LIN {X 0,Y 573.653,Z 410.287,A -85,B 0,C 180,E1 -2261.447,E2 -2261.447} C_VEL
LIN {X 0,Y 573.725,Z 397.169,A -85,B 0,C 180,E1 -2261.975,E2 -2261.975} C_VEL
LIN {X 0,Y 573.84,Z 384.516,A -85,B 0,C 180,E1 -2262.331,E2 -2262.331} C_VEL
LIN {X 0,Y 573.891,Z 371.307,A -85,B 0,C 180,E1 -2262.555,E2 -2262.555} C_VEL
LIN {X 0,Y 573.878,Z 274.271,A -85,B 0,C 180,E1 -2263.777,E2 -2263.777} C_VEL
LIN {X 0,Y 573.4,Z 270.792,A -85,B 0,C 180,E1 -2263.85,E2 -2263.85} C_VEL
LIN {X 0,Y 573.536,Z 250.898,A -85,B 0,C 180,E1 -2266.722,E2 -2266.722} C_VEL
LIN {X 0,Y 573.751,Z 233.17,A -85,B 0,C 180,E1 -2269.313,E2 -2269.313} C_VEL
LIN {X 0,Y 573.937,Z 214.032,A -85,B 0,C 180,E1 -2272.12,E2 -2272.12} C_VEL
LIN {X 0,Y 573.619,Z 210.185,A -85,B 0,C 180,E1 -2272.702,E2 -2272.702} C_VEL
LIN {X 0,Y 573.234,Z 208.084,A -85,B 0,C 180,E1 -2273.06,E2 -2273.06} C_VEL
LIN {X 0,Y 573.236,Z 208.085,A -85,B 0,C 180,E1 -2275.411,E2 -2275.411} C_VEL
LIN {X 0,Y 573.231,Z 208.076,A -85,B 0,C 180,E1 -2278.565,E2 -2278.565} C_VEL
LIN {X 0,Y 573.22,Z 208.08,A -85,B 0,C 180,E1 -2280.994,E2 -2280.994} C_VEL
LIN {X 0,Y 573.265,Z 208.081,A -85,B 0,C 180,E1 -2283.524,E2 -2283.524} C_VEL
LIN {X 0,Y 573.194,Z 208.082,A -85,B 0,C 180,E1 -2286.053,E2 -2286.053} C_VEL
LIN {X 0,Y 573.237,Z 208.075,A -85,B 0,C 180,E1 -2288.702,E2 -2288.702} C_VEL
LIN {X 0,Y 573.226,Z 208.084,A -85,B 0,C 180,E1 -2291.592,E2 -2291.592} C_VEL
LIN {X 0,Y 573.223,Z 208.076,A -85,B 0,C 180,E1 -2294.335,E2 -2294.335} C_VEL
LIN {X 0,Y 573.237,Z 208.083,A -85,B 0,C 180,E1 -2297.359,E2 -2297.359} C_VEL
LIN {X 0,Y 573.237,Z 208.074,A -85,B 0,C 180,E1 -2300.392,E2 -2300.392} C_VEL
LIN {X 0,Y 573.226,Z 208.079,A -85,B 0,C 180,E1 -2303.075,E2 -2303.075} C_VEL
LIN {X 0,Y 573.262,Z 208.077,A -85,B 0,C 180,E1 -2305.671,E2 -2305.671} C_VEL
LIN {X 0,Y 573.239,Z 208.075,A -85,B 0,C 180,E1 -2308.184,E2 -2308.184} C_VEL
LIN {X 0,Y 573.26,Z 208.071,A -85,B 0,C 180,E1 -2310.634,E2 -2310.634} C_VEL
LIN {X 0,Y 573.255,Z 208.075,A -85,B 0,C 180,E1 -2313.81,E2 -2313.81} C_VEL
LIN {X 0,Y 573.227,Z 208.076,A -85,B 0,C 180,E1 -2316.134,E2 -2316.134} C_VEL
LIN {X 0,Y 573.251,Z 208.077,A -85,B 0,C 180,E1 -2319.174,E2 -2319.174} C_VEL
LIN {X 0,Y 573.221,Z 208.086,A -85,B 0,C 180,E1 -2321.411,E2 -2321.411} C_VEL
LIN {X 0,Y 573.242,Z 208.08,A -85,B 0,C 180,E1 -2323.621,E2 -2323.621} C_VEL
LIN {X 0,Y 573.273,Z 208.074,A -85,B 0,C 180,E1 -2325.807,E2 -2325.807} C_VEL
LIN {X 0,Y 573.265,Z 208.071,A -85,B 0,C 180,E1 -2328.745,E2 -2328.745} C_VEL
LIN {X 0,Y 573.283,Z 208.076,A -85,B 0,C 180,E1 -2331.541,E2 -2331.541} C_VEL
LIN {X 0,Y 573.246,Z 208.079,A -85,B 0,C 180,E1 -2333.665,E2 -2333.665} C_VEL
LIN {X 0,Y 573.229,Z 208.079,A -85,B 0,C 180,E1 -2335.781,E2 -2335.781} C_VEL
LIN {X 0,Y 573.314,Z 208.067,A -85,B 0,C 180,E1 -2337.892,E2 -2337.892} C_VEL
LIN {X 0,Y 573.319,Z 208.065,A -85,B 0,C 180,E1 -2340.702,E2 -2340.702} C_VEL
LIN {X 0,Y 573.292,Z 208.068,A -85,B 0,C 180,E1 -2342.811,E2 -2342.811} C_VEL
LIN {X 0,Y 573.293,Z 208.074,A -85,B 0,C 180,E1 -2345.628,E2 -2345.628} C_VEL
LIN {X 0,Y 573.253,Z 208.071,A -85,B 0,C 180,E1 -2348.46,E2 -2348.46} C_VEL
LIN {X 0,Y 573.274,Z 208.078,A -85,B 0,C 180,E1 -2351.312,E2 -2351.312} C_VEL
LIN {X 0,Y 573.27,Z 208.07,A -85,B 0,C 180,E1 -2354.419,E2 -2354.419} C_VEL
LIN {X 0,Y 573.251,Z 208.077,A -85,B 0,C 180,E1 -2357.112,E2 -2357.112} C_VEL
LIN {X 0,Y 573.238,Z 208.075,A -85,B 0,C 180,E1 -2360.077,E2 -2360.077} C_VEL
LIN {X 0,Y 573.225,Z 208.074,A -85,B 0,C 180,E1 -2362.338,E2 -2362.338} C_VEL
LIN {X 0,Y 573.221,Z 208.076,A -85,B 0,C 180,E1 -2364.362,E2 -2364.362} C_VEL
LIN {X 0,Y 572.579,Z 208.16,A -85,B 0,C 180,E1 -2364.948,E2 -2364.948} C_VEL
LIN {X 0,Y 569.74,Z 208.519,A -85,B 0,C 180,E1 -2365.899,E2 -2365.899} C_VEL
LIN {X 0,Y 567.321,Z 208.823,A -85,B 0,C 180,E1 -2366.665,E2 -2366.665} C_VEL
LIN {X 0,Y 566.272,Z 208.95,A -85,B 0,C 180,E1 -2367.256,E2 -2367.256} C_VEL
LIN {X 0,Y 566.183,Z 208.959,A -85,B 0,C 180,E1 -2367.456,E2 -2367.456} C_VEL
LIN {X 0,Y 566.197,Z 208.955,A -85,B 0,C 180,E1 -2369.769,E2 -2369.769} C_VEL
LIN {X 0,Y 566.202,Z 208.951,A -85,B 0,C 180,E1 -2372.43,E2 -2372.43} C_VEL
LIN {X 0,Y 566.179,Z 208.957,A -85,B 0,C 180,E1 -2374.989,E2 -2374.989} C_VEL
LIN {X 0,Y 566.193,Z 208.961,A -85,B 0,C 180,E1 -2377.461,E2 -2377.461} C_VEL
LIN {X 0,Y 566.208,Z 208.95,A -85,B 0,C 180,E1 -2380.199,E2 -2380.199} C_VEL
LIN {X 0,Y 566.198,Z 208.956,A -85,B 0,C 180,E1 -2383.055,E2 -2383.055} C_VEL
LIN {X 0,Y 566.161,Z 208.956,A -85,B 0,C 180,E1 -2386.053,E2 -2386.053} C_VEL
LIN {X 0,Y 566.173,Z 208.958,A -85,B 0,C 180,E1 -2388.86,E2 -2388.86} C_VEL
LIN {X 0,Y 566.211,Z 208.96,A -85,B 0,C 180,E1 -2391.442,E2 -2391.442} C_VEL
LIN {X 0,Y 566.152,Z 208.958,A -85,B 0,C 180,E1 -2394.307,E2 -2394.307} C_VEL
LIN {X 0,Y 566.208,Z 208.953,A -85,B 0,C 180,E1 -2396.897,E2 -2396.897} C_VEL
LIN {X 0,Y 566.182,Z 208.962,A -85,B 0,C 180,E1 -2399.407,E2 -2399.407} C_VEL
LIN {X 0,Y 566.19,Z 208.956,A -85,B 0,C 180,E1 -2401.856,E2 -2401.856} C_VEL
LIN {X 0,Y 566.221,Z 209.027,A -85,B 0,C 180,E1 -2404.227,E2 -2404.227} C_VEL
LIN {X 0,Y 566.522,Z 213.688,A -85,B 0,C 180,E1 -2405.052,E2 -2405.052} C_VEL
LIN {X 0,Y 566.362,Z 230.218,A -85,B 0,C 180,E1 -2407.953,E2 -2407.953} C_VEL
LIN {X 0,Y 566.25,Z 242.171,A -85,B 0,C 180,E1 -2410.048,E2 -2410.048} C_VEL
LIN {X 0,Y 567.167,Z 248.554,A -85,B 0,C 180,E1 -2410.157,E2 -2410.157} C_VEL
LIN {X 0,Y 566.907,Z 349.31,A -85,B 0,C 180,E1 -2411.454,E2 -2411.454} C_VEL
LIN {X 0,Y 566.825,Z 362.732,A -85,B 0,C 180,E1 -2411.779,E2 -2411.779} C_VEL
LIN {X 0,Y 566.717,Z 375.02,A -85,B 0,C 180,E1 -2412.219,E2 -2412.219} C_VEL
LIN {X 0,Y 566.602,Z 386.826,A -85,B 0,C 180,E1 -2412.791,E2 -2412.791} C_VEL
LIN {X 0,Y 566.464,Z 398.37,A -85,B 0,C 180,E1 -2413.513,E2 -2413.513} C_VEL
LIN {X 0,Y 566.3,Z 408.957,A -85,B 0,C 180,E1 -2414.34,E2 -2414.34} C_VEL
LIN {X 0,Y 566.194,Z 418.423,A -85,B 0,C 180,E1 -2415.259,E2 -2415.259} C_VEL
LIN {X 0,Y 566.087,Z 427.544,A -85,B 0,C 180,E1 -2416.356,E2 -2416.356} C_VEL
LIN {X 0,Y 566.031,Z 434.851,A -85,B 0,C 180,E1 -2417.45,E2 -2417.45} C_VEL
LIN {X 0,Y 565.952,Z 440.637,A -85,B 0,C 180,E1 -2418.54,E2 -2418.54} C_VEL
LIN {X 0,Y 565.906,Z 445.169,A -85,B 0,C 180,E1 -2419.626,E2 -2419.626} C_VEL
LIN {X 0,Y 565.863,Z 448.594,A -85,B 0,C 180,E1 -2420.708,E2 -2420.708} C_VEL
LIN {X 0,Y 565.86,Z 450.288,A -85,B 0,C 180,E1 -2421.429,E2 -2421.429} C_VEL
LIN {X 0,Y 565.879,Z 451.573,A -85,B 0,C 180,E1 -2422.148,E2 -2422.148} C_VEL
LIN {X 0,Y 565.919,Z 452.869,A -85,B 0,C 180,E1 -2423.466,E2 -2423.466} C_VEL
LIN {X 0,Y 565.897,Z 452.951,A -85,B 0,C 180,E1 -2424.298,E2 -2424.298} C_VEL
LIN {X 0,Y 565.911,Z 451.892,A -85,B 0,C 180,E1 -2425.727,E2 -2425.727} C_VEL
LIN {X 0,Y 565.912,Z 450.734,A -85,B 0,C 180,E1 -2426.44,E2 -2426.44} C_VEL
LIN {X 0,Y 565.876,Z 449.165,A -85,B 0,C 180,E1 -2427.152,E2 -2427.152} C_VEL
LIN {X 0,Y 565.906,Z 446.016,A -85,B 0,C 180,E1 -2428.221,E2 -2428.221} C_VEL
LIN {X 0,Y 565.9,Z 441.822,A -85,B 0,C 180,E1 -2429.288,E2 -2429.288} C_VEL
LIN {X 0,Y 566.026,Z 435.459,A -85,B 0,C 180,E1 -2430.534,E2 -2430.534} C_VEL
LIN {X 0,Y 566.067,Z 428.544,A -85,B 0,C 180,E1 -2431.601,E2 -2431.601} C_VEL
LIN {X 0,Y 566.142,Z 419.905,A -85,B 0,C 180,E1 -2432.668,E2 -2432.668} C_VEL
LIN {X 0,Y 566.241,Z 411.087,A -85,B 0,C 180,E1 -2433.558,E2 -2433.558} C_VEL
LIN {X 0,Y 566.404,Z 400.228,A -85,B 0,C 180,E1 -2434.448,E2 -2434.448} C_VEL
LIN {X 0,Y 566.585,Z 389.269,A -85,B 0,C 180,E1 -2435.16,E2 -2435.16} C_VEL
LIN {X 0,Y 566.686,Z 377.045,A -85,B 0,C 180,E1 -2435.783,E2 -2435.783} C_VEL
LIN {X 0,Y 566.844,Z 365.434,A -85,B 0,C 180,E1 -2436.228,E2 -2436.228} C_VEL
LIN {X 0,Y 566.944,Z 352.308,A -85,B 0,C 180,E1 -2436.575,E2 -2436.575} C_VEL
LIN {X 0,Y 567.009,Z 333.787,A -85,B 0,C 180,E1 -2436.85,E2 -2436.85} C_VEL
LIN {X 0,Y 567.123,Z 247.443,A -85,B 0,C 180,E1 -2437.948,E2 -2437.948} C_VEL
LIN {X 0,Y 566.253,Z 242.163,A -85,B 0,C 180,E1 -2438.043,E2 -2438.043} C_VEL
LIN {X 0,Y 566.444,Z 224.855,A -85,B 0,C 180,E1 -2441.083,E2 -2441.083} C_VEL
LIN {X 0,Y 566.545,Z 211.416,A -85,B 0,C 180,E1 -2443.45,E2 -2443.45} C_VEL
LIN {X 0,Y 566.232,Z 208.954,A -85,B 0,C 180,E1 -2443.915,E2 -2443.915} C_VEL
LIN {X 0,Y 566.229,Z 208.952,A -85,B 0,C 180,E1 -2447.113,E2 -2447.113} C_VEL
LIN {X 0,Y 566.206,Z 208.95,A -85,B 0,C 180,E1 -2449.581,E2 -2449.581} C_VEL
LIN {X 0,Y 566.196,Z 208.951,A -85,B 0,C 180,E1 -2451.862,E2 -2451.862} C_VEL
LIN {X 0,Y 566.222,Z 208.952,A -85,B 0,C 180,E1 -2455.03,E2 -2455.03} C_VEL
LIN {X 0,Y 566.176,Z 208.955,A -85,B 0,C 180,E1 -2457.341,E2 -2457.341} C_VEL
LIN {X 0,Y 566.203,Z 208.95,A -85,B 0,C 180,E1 -2459.769,E2 -2459.769} C_VEL
LIN {X 0,Y 566.205,Z 208.956,A -85,B 0,C 180,E1 -2462.429,E2 -2462.429} C_VEL
LIN {X 0,Y 566.182,Z 208.958,A -85,B 0,C 180,E1 -2464.989,E2 -2464.989} C_VEL
LIN {X 0,Y 566.194,Z 208.952,A -85,B 0,C 180,E1 -2467.461,E2 -2467.461} C_VEL
LIN {X 0,Y 566.209,Z 208.953,A -85,B 0,C 180,E1 -2470.199,E2 -2470.199} C_VEL
LIN {X 0,Y 566.199,Z 208.955,A -85,B 0,C 180,E1 -2473.054,E2 -2473.054} C_VEL
LIN {X 0,Y 566.195,Z 208.953,A -85,B 0,C 180,E1 -2476.049,E2 -2476.049} C_VEL
LIN {X 0,Y 566.205,Z 208.952,A -85,B 0,C 180,E1 -2479.214,E2 -2479.214} C_VEL
LIN {X 0,Y 566.183,Z 208.953,A -85,B 0,C 180,E1 -2481.636,E2 -2481.636} C_VEL
LIN {X 0,Y 566.151,Z 208.961,A -85,B 0,C 180,E1 -2484.307,E2 -2484.307} C_VEL
LIN {X 0,Y 566.221,Z 208.954,A -85,B 0,C 180,E1 -2486.898,E2 -2486.898} C_VEL
LIN {X 0,Y 566.18,Z 208.954,A -85,B 0,C 180,E1 -2489.407,E2 -2489.407} C_VEL
LIN {X 0,Y 566.192,Z 208.952,A -85,B 0,C 180,E1 -2491.856,E2 -2491.856} C_VEL
LIN {X 0,Y 566.196,Z 208.955,A -85,B 0,C 180,E1 -2494.25,E2 -2494.25} C_VEL
LIN {X 0,Y 566.171,Z 208.963,A -85,B 0,C 180,E1 -2496.719,E2 -2496.719} C_VEL
LIN {X 0,Y 566.205,Z 208.95,A -85,B 0,C 180,E1 -2499.662,E2 -2499.662} C_VEL
LIN {X 0,Y 566.2,Z 208.961,A -85,B 0,C 180,E1 -2502.668,E2 -2502.668} C_VEL
LIN {X 0,Y 566.222,Z 208.948,A -85,B 0,C 180,E1 -2505.626,E2 -2505.626} C_VEL
LIN {X 0,Y 566.236,Z 208.956,A -85,B 0,C 180,E1 -2508.675,E2 -2508.675} C_VEL
LIN {X 0,Y 566.204,Z 208.95,A -85,B 0,C 180,E1 -2511.434,E2 -2511.434} C_VEL
LIN {X 0,Y 566.262,Z 208.948,A -85,B 0,C 180,E1 -2514.302,E2 -2514.302} C_VEL
LIN {X 0,Y 566.282,Z 208.941,A -85,B 0,C 180,E1 -2517.866,E2 -2517.866} C_VEL
LIN {X 0,Y 566.302,Z 208.947,A -85,B 0,C 180,E1 -2520.711,E2 -2520.711} C_VEL
LIN {X 0,Y 566.27,Z 208.948,A -85,B 0,C 180,E1 -2522.846,E2 -2522.846} C_VEL
LIN {X 0,Y 566.25,Z 208.945,A -85,B 0,C 180,E1 -2525.698,E2 -2525.698} C_VEL
LIN {X 0,Y 566.226,Z 208.957,A -85,B 0,C 180,E1 -2528.566,E2 -2528.566} C_VEL
LIN {X 0,Y 566.243,Z 208.945,A -85,B 0,C 180,E1 -2531.454,E2 -2531.454} C_VEL
LIN {X 0,Y 566.235,Z 208.955,A -85,B 0,C 180,E1 -2534.506,E2 -2534.506} C_VEL
LIN {X 0,Y 566.194,Z 208.952,A -85,B 0,C 180,E1 -2537.332,E2 -2537.332} C_VEL
LIN {X 0,Y 566.207,Z 208.956,A -85,B 0,C 180,E1 -2540.337,E2 -2540.337} C_VEL
LIN {X 0,Y 566.169,Z 208.955,A -85,B 0,C 180,E1 -2543.281,E2 -2543.281} C_VEL
LIN {X 0,Y 566.205,Z 208.95,A -85,B 0,C 180,E1 -2545.749,E2 -2545.749} C_VEL
LIN {X 0,Y 566.185,Z 208.957,A -85,B 0,C 180,E1 -2548.954,E2 -2548.954} C_VEL
LIN {X 0,Y 566.192,Z 208.952,A -85,B 0,C 180,E1 -2551.422,E2 -2551.422} C_VEL
LIN {X 0,Y 566.201,Z 208.952,A -85,B 0,C 180,E1 -2553.957,E2 -2553.957} C_VEL
LIN {X 0,Y 566.182,Z 208.963,A -85,B 0,C 180,E1 -2556.571,E2 -2556.571} C_VEL
LIN {X 0,Y 566.212,Z 208.95,A -85,B 0,C 180,E1 -2559.274,E2 -2559.274} C_VEL
LIN {X 0,Y 566.188,Z 208.955,A -85,B 0,C 180,E1 -2562.09,E2 -2562.09} C_VEL
LIN {X 0,Y 566.165,Z 208.958,A -85,B 0,C 180,E1 -2565.037,E2 -2565.037} C_VEL
LIN {X 0,Y 566.187,Z 208.954,A -85,B 0,C 180,E1 -2567.91,E2 -2567.91} C_VEL
LIN {X 0,Y 566.211,Z 208.956,A -85,B 0,C 180,E1 -2570.726,E2 -2570.726} C_VEL
LIN {X 0,Y 566.182,Z 208.953,A -85,B 0,C 180,E1 -2573.429,E2 -2573.429} C_VEL
LIN {X 0,Y 566.213,Z 208.955,A -85,B 0,C 180,E1 -2576.266,E2 -2576.266} C_VEL
LIN {X 0,Y 566.186,Z 208.956,A -85,B 0,C 180,E1 -2578.925,E2 -2578.925} C_VEL
LIN {X 0,Y 566.192,Z 208.954,A -85,B 0,C 180,E1 -2581.856,E2 -2581.856} C_VEL
LIN {X 0,Y 566.196,Z 208.958,A -85,B 0,C 180,E1 -2584.25,E2 -2584.25} C_VEL
LIN {X 0,Y 566.21,Z 209.141,A -85,B 0,C 180,E1 -2586.852,E2 -2586.852} C_VEL
LIN {X 0,Y 567.008,Z 213.862,A -85,B 0,C 180,E1 -2587.596,E2 -2587.596} C_VEL
LIN {X 0,Y 566.766,Z 233.934,A -85,B 0,C 180,E1 -2590.578,E2 -2590.578} C_VEL
LIN {X 0,Y 566.551,Z 252.227,A -85,B 0,C 180,E1 -2593.262,E2 -2593.262} C_VEL
LIN {X 0,Y 566.418,Z 271.144,A -85,B 0,C 180,E1 -2595.998,E2 -2595.998} C_VEL
LIN {X 0,Y 567.165,Z 276.51,A -85,B 0,C 180,E1 -2596.086,E2 -2596.086} C_VEL
LIN {X 0,Y 566.918,Z 378.947,A -85,B 0,C 180,E1 -2597.402,E2 -2597.402} C_VEL
LIN {X 0,Y 566.839,Z 392.218,A -85,B 0,C 180,E1 -2597.719,E2 -2597.719} C_VEL
LIN {X 0,Y 566.724,Z 404.378,A -85,B 0,C 180,E1 -2598.148,E2 -2598.148} C_VEL
LIN {X 0,Y 566.603,Z 416.367,A -85,B 0,C 180,E1 -2598.72,E2 -2598.72} C_VEL
LIN {X 0,Y 566.45,Z 428.197,A -85,B 0,C 180,E1 -2599.455,E2 -2599.455} C_VEL
LIN {X 0,Y 566.324,Z 438.604,A -85,B 0,C 180,E1 -2600.265,E2 -2600.265} C_VEL
LIN {X 0,Y 566.207,Z 447.113,A -85,B 0,C 180,E1 -2601.074,E2 -2601.074} C_VEL
LIN {X 0,Y 566.112,Z 454.961,A -85,B 0,C 180,E1 -2601.972,E2 -2601.972} C_VEL
LIN {X 0,Y 566.003,Z 462.622,A -85,B 0,C 180,E1 -2603.047,E2 -2603.047} C_VEL
LIN {X 0,Y 566.004,Z 469.68,A -85,B 0,C 180,E1 -2604.299,E2 -2604.299} C_VEL
LIN {X 0,Y 565.933,Z 474.373,A -85,B 0,C 180,E1 -2605.37,E2 -2605.37} C_VEL
LIN {X 0,Y 565.927,Z 477.958,A -85,B 0,C 180,E1 -2606.44,E2 -2606.44} C_VEL
LIN {X 0,Y 565.878,Z 479.808,A -85,B 0,C 180,E1 -2607.152,E2 -2607.152} C_VEL
LIN {X 0,Y 565.846,Z 482.184,A -85,B 0,C 180,E1 -2608.577,E2 -2608.577} C_VEL
LIN {X 0,Y 565.839,Z 483,A -85,B 0,C 180,E1 -2610,E2 -2610} C_VEL
LIN {X 0,Y 565.846,Z 482.185,A -85,B 0,C 180,E1 -2611.423,E2 -2611.423} C_VEL
LIN {X 0,Y 565.878,Z 479.81,A -85,B 0,C 180,E1 -2612.848,E2 -2612.848} C_VEL
LIN {X 0,Y 565.926,Z 476.895,A -85,B 0,C 180,E1 -2613.917,E2 -2613.917} C_VEL
LIN {X 0,Y 565.878,Z 472.948,A -85,B 0,C 180,E1 -2614.987,E2 -2614.987} C_VEL
LIN {X 0,Y 566.002,Z 467.867,A -85,B 0,C 180,E1 -2616.059,E2 -2616.059} C_VEL
LIN {X 0,Y 566.04,Z 461.467,A -85,B 0,C 180,E1 -2617.132,E2 -2617.132} C_VEL
LIN {X 0,Y 566.134,Z 453.477,A -85,B 0,C 180,E1 -2618.208,E2 -2618.208} C_VEL
LIN {X 0,Y 566.229,Z 445.334,A -85,B 0,C 180,E1 -2619.105,E2 -2619.105} C_VEL
LIN {X 0,Y 566.345,Z 435.399,A -85,B 0,C 180,E1 -2620.005,E2 -2620.005} C_VEL
LIN {X 0,Y 566.529,Z 424.303,A -85,B 0,C 180,E1 -2620.807,E2 -2620.807} C_VEL
LIN {X 0,Y 566.613,Z 413.173,A -85,B 0,C 180,E1 -2621.447,E2 -2621.447} C_VEL
LIN {X 0,Y 566.723,Z 400.979,A -85,B 0,C 180,E1 -2621.989,E2 -2621.989} C_VEL
LIN {X 0,Y 566.852,Z 388.173,A -85,B 0,C 180,E1 -2622.395,E2 -2622.395} C_VEL
LIN {X 0,Y 566.978,Z 374.598,A -85,B 0,C 180,E1 -2622.665,E2 -2622.665} C_VEL
LIN {X 0,Y 567.043,Z 275.419,A -85,B 0,C 180,E1 -2623.931,E2 -2623.931} C_VEL
LIN {X 0,Y 566.396,Z 270.792,A -85,B 0,C 180,E1 -2624.025,E2 -2624.025} C_VEL
LIN {X 0,Y 566.569,Z 249.762,A -85,B 0,C 180,E1 -2627.101,E2 -2627.101} C_VEL
LIN {X 0,Y 566.78,Z 231.71,A -85,B 0,C 180,E1 -2629.749,E2 -2629.749} C_VEL
LIN {X 0,Y 567.007,Z 213.826,A -85,B 0,C 180,E1 -2632.405,E2 -2632.405} C_VEL
LIN {X 0,Y 566.176,Z 208.964,A -85,B 0,C 180,E1 -2633.201,E2 -2633.201} C_VEL
LIN {X 0,Y 566.196,Z 208.959,A -85,B 0,C 180,E1 -2635.75,E2 -2635.75} C_VEL
LIN {X 0,Y 566.205,Z 208.953,A -85,B 0,C 180,E1 -2638.202,E2 -2638.202} C_VEL
LIN {X 0,Y 566.186,Z 208.957,A -85,B 0,C 180,E1 -2641.075,E2 -2641.075} C_VEL
LIN {X 0,Y 566.213,Z 208.955,A -85,B 0,C 180,E1 -2643.734,E2 -2643.734} C_VEL
LIN {X 0,Y 566.182,Z 208.953,A -85,B 0,C 180,E1 -2646.571,E2 -2646.571} C_VEL
LIN {X 0,Y 566.214,Z 208.956,A -85,B 0,C 180,E1 -2649.685,E2 -2649.685} C_VEL
LIN {X 0,Y 566.197,Z 208.954,A -85,B 0,C 180,E1 -2652.916,E2 -2652.916} C_VEL
LIN {X 0,Y 566.16,Z 208.959,A -85,B 0,C 180,E1 -2655.96,E2 -2655.96} C_VEL
LIN {X 0,Y 566.186,Z 208.954,A -85,B 0,C 180,E1 -2658.14,E2 -2658.14} C_VEL
LIN {X 0,Y 566.212,Z 208.95,A -85,B 0,C 180,E1 -2660.726,E2 -2660.726} C_VEL
LIN {X 0,Y 566.178,Z 208.963,A -85,B 0,C 180,E1 -2663.428,E2 -2663.428} C_VEL
LIN {X 0,Y 566.198,Z 208.95,A -85,B 0,C 180,E1 -2666.268,E2 -2666.268} C_VEL
LIN {X 0,Y 566.189,Z 208.954,A -85,B 0,C 180,E1 -2668.924,E2 -2668.924} C_VEL
LIN {X 0,Y 566.188,Z 208.956,A -85,B 0,C 180,E1 -2671.856,E2 -2671.856} C_VEL
LIN {X 0,Y 566.205,Z 208.949,A -85,B 0,C 180,E1 -2674.251,E2 -2674.251} C_VEL
LIN {X 0,Y 566.169,Z 208.956,A -85,B 0,C 180,E1 -2676.719,E2 -2676.719} C_VEL
LIN {X 0,Y 566.208,Z 208.956,A -85,B 0,C 180,E1 -2679.663,E2 -2679.663} C_VEL
LIN {X 0,Y 566.195,Z 208.951,A -85,B 0,C 180,E1 -2682.668,E2 -2682.668} C_VEL
LIN {X 0,Y 566.235,Z 208.953,A -85,B 0,C 180,E1 -2685.627,E2 -2685.627} C_VEL
LIN {X 0,Y 566.236,Z 208.946,A -85,B 0,C 180,E1 -2688.675,E2 -2688.675} C_VEL
LIN {X 0,Y 566.226,Z 208.957,A -85,B 0,C 180,E1 -2691.434,E2 -2691.434} C_VEL
LIN {X 0,Y 566.249,Z 208.944,A -85,B 0,C 180,E1 -2694.302,E2 -2694.302} C_VEL
LIN {X 0,Y 566.284,Z 208.942,A -85,B 0,C 180,E1 -2697.866,E2 -2697.866} C_VEL
LIN {X 0,Y 566.291,Z 208.94,A -85,B 0,C 180,E1 -2700.711,E2 -2700.711} C_VEL
LIN {X 0,Y 566.26,Z 208.944,A -85,B 0,C 180,E1 -2702.846,E2 -2702.846} C_VEL
LIN {X 0,Y 566.26,Z 208.949,A -85,B 0,C 180,E1 -2705.698,E2 -2705.698} C_VEL
LIN {X 0,Y 566.204,Z 208.949,A -85,B 0,C 180,E1 -2708.566,E2 -2708.566} C_VEL
LIN {X 0,Y 566.244,Z 208.955,A -85,B 0,C 180,E1 -2711.454,E2 -2711.454} C_VEL
LIN {X 0,Y 566.225,Z 208.947,A -85,B 0,C 180,E1 -2714.502,E2 -2714.502} C_VEL
LIN {X 0,Y 566.193,Z 208.96,A -85,B 0,C 180,E1 -2717.332,E2 -2717.332} C_VEL
LIN {X 0,Y 566.205,Z 208.95,A -85,B 0,C 180,E1 -2720.338,E2 -2720.338} C_VEL
LIN {X 0,Y 566.169,Z 208.961,A -85,B 0,C 180,E1 -2723.281,E2 -2723.281} C_VEL
LIN {X 0,Y 566.196,Z 208.955,A -85,B 0,C 180,E1 -2725.75,E2 -2725.75} C_VEL
LIN {X 0,Y 566.183,Z 208.959,A -85,B 0,C 180,E1 -2727.456,E2 -2727.456} C_VEL
LIN {X 0,Y 565.504,Z 209.04,A -85,B 0,C 180,E1 -2728.05,E2 -2728.05} C_VEL
LIN {X 0,Y 562.646,Z 209.397,A -85,B 0,C 180,E1 -2729.014,E2 -2729.014} C_VEL
LIN {X 0,Y 560.242,Z 209.696,A -85,B 0,C 180,E1 -2729.79,E2 -2729.79} C_VEL
LIN {X 0,Y 559.216,Z 209.82,A -85,B 0,C 180,E1 -2730.389,E2 -2730.389} C_VEL
LIN {X 0,Y 559.136,Z 209.83,A -85,B 0,C 180,E1 -2730.591,E2 -2730.591} C_VEL
LIN {X 0,Y 559.158,Z 209.829,A -85,B 0,C 180,E1 -2732.715,E2 -2732.715} C_VEL
LIN {X 0,Y 559.124,Z 209.841,A -85,B 0,C 180,E1 -2735.325,E2 -2735.325} C_VEL
LIN {X 0,Y 559.131,Z 209.833,A -85,B 0,C 180,E1 -2738.018,E2 -2738.018} C_VEL
LIN {X 0,Y 559.157,Z 209.83,A -85,B 0,C 180,E1 -2740.813,E2 -2740.813} C_VEL
LIN {X 0,Y 559.138,Z 209.836,A -85,B 0,C 180,E1 -2743.735,E2 -2743.735} C_VEL
LIN {X 0,Y 559.133,Z 209.832,A -85,B 0,C 180,E1 -2746.805,E2 -2746.805} C_VEL
LIN {X 0,Y 559.157,Z 209.836,A -85,B 0,C 180,E1 -2749.188,E2 -2749.188} C_VEL
LIN {X 0,Y 559.133,Z 209.834,A -85,B 0,C 180,E1 -2751.982,E2 -2751.982} C_VEL
LIN {X 0,Y 559.131,Z 209.835,A -85,B 0,C 180,E1 -2754.788,E2 -2754.788} C_VEL
LIN {X 0,Y 559.157,Z 209.838,A -85,B 0,C 180,E1 -2757.365,E2 -2757.365} C_VEL
LIN {X 0,Y 559.15,Z 209.829,A -85,B 0,C 180,E1 -2760.143,E2 -2760.143} C_VEL
LIN {X 0,Y 559.163,Z 209.835,A -85,B 0,C 180,E1 -2763.175,E2 -2763.175} C_VEL
LIN {X 0,Y 559.192,Z 209.931,A -85,B 0,C 180,E1 -2764.154,E2 -2764.154} C_VEL
LIN {X 0,Y 559.513,Z 215.396,A -85,B 0,C 180,E1 -2765.127,E2 -2765.127} C_VEL
LIN {X 0,Y 559.348,Z 230.858,A -85,B 0,C 180,E1 -2767.856,E2 -2767.856} C_VEL
LIN {X 0,Y 559.214,Z 242.153,A -85,B 0,C 180,E1 -2769.862,E2 -2769.862} C_VEL
LIN {X 0,Y 560.285,Z 249.022,A -85,B 0,C 180,E1 -2769.989,E2 -2769.989} C_VEL
LIN {X 0,Y 560.001,Z 348.905,A -85,B 0,C 180,E1 -2771.288,E2 -2771.288} C_VEL
LIN {X 0,Y 559.891,Z 362.454,A -85,B 0,C 180,E1 -2771.616,E2 -2771.616} C_VEL
LIN {X 0,Y 559.764,Z 375.39,A -85,B 0,C 180,E1 -2772.085,E2 -2772.085} C_VEL
LIN {X 0,Y 559.627,Z 387.102,A -85,B 0,C 180,E1 -2772.665,E2 -2772.665} C_VEL
LIN {X 0,Y 559.455,Z 398.577,A -85,B 0,C 180,E1 -2773.394,E2 -2773.394} C_VEL
LIN {X 0,Y 559.278,Z 409.13,A -85,B 0,C 180,E1 -2774.232,E2 -2774.232} C_VEL
LIN {X 0,Y 559.173,Z 417.716,A -85,B 0,C 180,E1 -2775.069,E2 -2775.069} C_VEL
LIN {X 0,Y 559.056,Z 425.638,A -85,B 0,C 180,E1 -2776.003,E2 -2776.003} C_VEL
LIN {X 0,Y 558.937,Z 433.241,A -85,B 0,C 180,E1 -2777.104,E2 -2777.104} C_VEL
LIN {X 0,Y 558.868,Z 440.281,A -85,B 0,C 180,E1 -2778.392,E2 -2778.392} C_VEL
LIN {X 0,Y 558.831,Z 444.901,A -85,B 0,C 180,E1 -2779.493,E2 -2779.493} C_VEL
LIN {X 0,Y 558.783,Z 448.396,A -85,B 0,C 180,E1 -2780.59,E2 -2780.59} C_VEL
LIN {X 0,Y 558.777,Z 450.134,A -85,B 0,C 180,E1 -2781.319,E2 -2781.319} C_VEL
LIN {X 0,Y 558.798,Z 451.454,A -85,B 0,C 180,E1 -2782.048,E2 -2782.048} C_VEL
LIN {X 0,Y 558.847,Z 452.872,A -85,B 0,C 180,E1 -2783.464,E2 -2783.464} C_VEL
LIN {X 0,Y 558.809,Z 452.967,A -85,B 0,C 180,E1 -2784.225,E2 -2784.225} C_VEL
LIN {X 0,Y 558.803,Z 451.977,A -85,B 0,C 180,E1 -2785.672,E2 -2785.672} C_VEL
LIN {X 0,Y 558.821,Z 450.884,A -85,B 0,C 180,E1 -2786.395,E2 -2786.395} C_VEL
LIN {X 0,Y 558.797,Z 449.351,A -85,B 0,C 180,E1 -2787.116,E2 -2787.116} C_VEL
LIN {X 0,Y 558.822,Z 446.275,A -85,B 0,C 180,E1 -2788.198,E2 -2788.198} C_VEL
LIN {X 0,Y 558.807,Z 442.16,A -85,B 0,C 180,E1 -2789.279,E2 -2789.279} C_VEL
LIN {X 0,Y 558.943,Z 435.882,A -85,B 0,C 180,E1 -2790.54,E2 -2790.54} C_VEL
LIN {X 0,Y 558.999,Z 429.07,A -85,B 0,C 180,E1 -2791.621,E2 -2791.621} C_VEL
LIN {X 0,Y 559.092,Z 420.583,A -85,B 0,C 180,E1 -2792.702,E2 -2792.702} C_VEL
LIN {X 0,Y 559.198,Z 411.898,A -85,B 0,C 180,E1 -2793.603,E2 -2793.603} C_VEL
LIN {X 0,Y 559.395,Z 401.229,A -85,B 0,C 180,E1 -2794.504,E2 -2794.504} C_VEL
LIN {X 0,Y 559.573,Z 390.578,A -85,B 0,C 180,E1 -2795.224,E2 -2795.224} C_VEL
LIN {X 0,Y 559.695,Z 378.691,A -85,B 0,C 180,E1 -2795.856,E2 -2795.856} C_VEL
LIN {X 0,Y 559.896,Z 366.302,A -85,B 0,C 180,E1 -2796.351,E2 -2796.351} C_VEL
LIN {X 0,Y 560.002,Z 353.377,A -85,B 0,C 180,E1 -2796.712,E2 -2796.712} C_VEL
LIN {X 0,Y 560.079,Z 337.813,A -85,B 0,C 180,E1 -2796.96,E2 -2796.96} C_VEL
LIN {X 0,Y 560.286,Z 248.574,A -85,B 0,C 180,E1 -2798.107,E2 -2798.107} C_VEL
LIN {X 0,Y 559.266,Z 242.169,A -85,B 0,C 180,E1 -2798.223,E2 -2798.223} C_VEL
LIN {X 0,Y 559.451,Z 225.478,A -85,B 0,C 180,E1 -2801.189,E2 -2801.189} C_VEL
LIN {X 0,Y 559.495,Z 211.794,A -85,B 0,C 180,E1 -2803.623,E2 -2803.623} C_VEL
LIN {X 0,Y 559.193,Z 209.831,A -85,B 0,C 180,E1 -2804.001,E2 -2804.001} C_VEL
LIN {X 0,Y 559.176,Z 209.83,A -85,B 0,C 180,E1 -2807.213,E2 -2807.213} C_VEL
LIN {X 0,Y 559.169,Z 209.827,A -85,B 0,C 180,E1 -2809.837,E2 -2809.837} C_VEL
LIN {X 0,Y 559.144,Z 209.832,A -85,B 0,C 180,E1 -2812.153,E2 -2812.153} C_VEL
LIN {X 0,Y 559.178,Z 209.827,A -85,B 0,C 180,E1 -2815.298,E2 -2815.298} C_VEL
LIN {X 0,Y 559.131,Z 209.831,A -85,B 0,C 180,E1 -2817.715,E2 -2817.715} C_VEL
LIN {X 0,Y 559.155,Z 209.831,A -85,B 0,C 180,E1 -2820.183,E2 -2820.183} C_VEL
LIN {X 0,Y 559.156,Z 209.838,A -85,B 0,C 180,E1 -2822.715,E2 -2822.715} C_VEL
LIN {X 0,Y 559.126,Z 209.833,A -85,B 0,C 180,E1 -2825.324,E2 -2825.324} C_VEL
LIN {X 0,Y 559.133,Z 209.832,A -85,B 0,C 180,E1 -2828.018,E2 -2828.018} C_VEL
LIN {X 0,Y 559.157,Z 209.836,A -85,B 0,C 180,E1 -2830.812,E2 -2830.812} C_VEL
LIN {X 0,Y 559.139,Z 209.83,A -85,B 0,C 180,E1 -2833.734,E2 -2833.734} C_VEL
LIN {X 0,Y 559.143,Z 209.837,A -85,B 0,C 180,E1 -2836.804,E2 -2836.804} C_VEL
LIN {X 0,Y 559.157,Z 209.83,A -85,B 0,C 180,E1 -2839.187,E2 -2839.187} C_VEL
LIN {X 0,Y 559.131,Z 209.832,A -85,B 0,C 180,E1 -2841.982,E2 -2841.982} C_VEL
LIN {X 0,Y 559.13,Z 209.839,A -85,B 0,C 180,E1 -2844.787,E2 -2844.787} C_VEL
LIN {X 0,Y 559.156,Z 209.829,A -85,B 0,C 180,E1 -2847.364,E2 -2847.364} C_VEL
LIN {X 0,Y 559.148,Z 209.832,A -85,B 0,C 180,E1 -2850.143,E2 -2850.143} C_VEL
LIN {X 0,Y 559.16,Z 209.83,A -85,B 0,C 180,E1 -2853.175,E2 -2853.175} C_VEL
LIN {X 0,Y 559.128,Z 209.832,A -85,B 0,C 180,E1 -2855.493,E2 -2855.493} C_VEL
LIN {X 0,Y 559.173,Z 209.836,A -85,B 0,C 180,E1 -2858.624,E2 -2858.624} C_VEL
LIN {X 0,Y 559.161,Z 209.833,A -85,B 0,C 180,E1 -2860.926,E2 -2860.926} C_VEL
LIN {X 0,Y 559.157,Z 209.829,A -85,B 0,C 180,E1 -2863.947,E2 -2863.947} C_VEL
LIN {X 0,Y 559.164,Z 209.83,A -85,B 0,C 180,E1 -2866.184,E2 -2866.184} C_VEL
LIN {X 0,Y 559.193,Z 209.826,A -85,B 0,C 180,E1 -2869.133,E2 -2869.133} C_VEL
LIN {X 0,Y 559.196,Z 209.825,A -85,B 0,C 180,E1 -2872.053,E2 -2872.053} C_VEL
LIN {X 0,Y 559.246,Z 209.821,A -85,B 0,C 180,E1 -2874.953,E2 -2874.953} C_VEL
LIN {X 0,Y 559.253,Z 209.817,A -85,B 0,C 180,E1 -2877.839,E2 -2877.839} C_VEL
LIN {X 0,Y 559.272,Z 209.822,A -85,B 0,C 180,E1 -2880.72,E2 -2880.72} C_VEL
LIN {X 0,Y 559.236,Z 209.824,A -85,B 0,C 180,E1 -2882.881,E2 -2882.881} C_VEL
LIN {X 0,Y 559.221,Z 209.82,A -85,B 0,C 180,E1 -2885.77,E2 -2885.77} C_VEL
LIN {X 0,Y 559.185,Z 209.833,A -85,B 0,C 180,E1 -2888.674,E2 -2888.674} C_VEL
LIN {X 0,Y 559.206,Z 209.822,A -85,B 0,C 180,E1 -2891.6,E2 -2891.6} C_VEL
LIN {X 0,Y 559.202,Z 209.833,A -85,B 0,C 180,E1 -2894.595,E2 -2894.595} C_VEL
LIN {X 0,Y 559.138,Z 209.83,A -85,B 0,C 180,E1 -2897.558,E2 -2897.558} C_VEL
LIN {X 0,Y 559.166,Z 209.828,A -85,B 0,C 180,E1 -2899.838,E2 -2899.838} C_VEL
LIN {X 0,Y 559.14,Z 209.834,A -85,B 0,C 180,E1 -2902.153,E2 -2902.153} C_VEL
LIN {X 0,Y 559.175,Z 209.827,A -85,B 0,C 180,E1 -2905.298,E2 -2905.298} C_VEL
LIN {X 0,Y 559.127,Z 209.832,A -85,B 0,C 180,E1 -2907.715,E2 -2907.715} C_VEL
LIN {X 0,Y 559.152,Z 209.833,A -85,B 0,C 180,E1 -2910.183,E2 -2910.183} C_VEL
LIN {X 0,Y 559.153,Z 209.836,A -85,B 0,C 180,E1 -2912.716,E2 -2912.716} C_VEL
LIN {X 0,Y 559.123,Z 209.833,A -85,B 0,C 180,E1 -2915.325,E2 -2915.325} C_VEL
LIN {X 0,Y 559.131,Z 209.833,A -85,B 0,C 180,E1 -2918.018,E2 -2918.018} C_VEL
LIN {X 0,Y 559.155,Z 209.834,A -85,B 0,C 180,E1 -2920.813,E2 -2920.813} C_VEL
LIN {X 0,Y 559.111,Z 209.834,A -85,B 0,C 180,E1 -2923.737,E2 -2923.737} C_VEL
LIN {X 0,Y 559.137,Z 209.836,A -85,B 0,C 180,E1 -2926.266,E2 -2926.266} C_VEL
LIN {X 0,Y 559.156,Z 209.829,A -85,B 0,C 180,E1 -2929.188,E2 -2929.188} C_VEL
LIN {X 0,Y 559.129,Z 209.833,A -85,B 0,C 180,E1 -2931.982,E2 -2931.982} C_VEL
LIN {X 0,Y 559.129,Z 209.837,A -85,B 0,C 180,E1 -2934.788,E2 -2934.788} C_VEL
LIN {X 0,Y 559.156,Z 209.828,A -85,B 0,C 180,E1 -2937.365,E2 -2937.365} C_VEL
LIN {X 0,Y 559.144,Z 209.834,A -85,B 0,C 180,E1 -2940.144,E2 -2940.144} C_VEL
LIN {X 0,Y 559.16,Z 209.831,A -85,B 0,C 180,E1 -2943.175,E2 -2943.175} C_VEL
LIN {X 0,Y 559.126,Z 209.833,A -85,B 0,C 180,E1 -2945.494,E2 -2945.494} C_VEL
LIN {X 0,Y 559.141,Z 209.904,A -85,B 0,C 180,E1 -2946.688,E2 -2946.688} C_VEL
LIN {X 0,Y 560.031,Z 214.953,A -85,B 0,C 180,E1 -2947.496,E2 -2947.496} C_VEL
LIN {X 0,Y 559.811,Z 233.681,A -85,B 0,C 180,E1 -2950.317,E2 -2950.317} C_VEL
LIN {X 0,Y 559.544,Z 251.326,A -85,B 0,C 180,E1 -2952.933,E2 -2952.933} C_VEL
LIN {X 0,Y 559.409,Z 271.144,A -85,B 0,C 180,E1 -2955.819,E2 -2955.819} C_VEL
LIN {X 0,Y 560.283,Z 278.299,A -85,B 0,C 180,E1 -2955.934,E2 -2955.934} C_VEL
LIN {X 0,Y 560.015,Z 378.947,A -85,B 0,C 180,E1 -2957.244,E2 -2957.244} C_VEL
LIN {X 0,Y 559.894,Z 392.218,A -85,B 0,C 180,E1 -2957.564,E2 -2957.564} C_VEL
LIN {X 0,Y 559.767,Z 404.378,A -85,B 0,C 180,E1 -2957.998,E2 -2957.998} C_VEL
LIN {X 0,Y 559.629,Z 416.194,A -85,B 0,C 180,E1 -2958.567,E2 -2958.567} C_VEL
LIN {X 0,Y 559.457,Z 428.195,A -85,B 0,C 180,E1 -2959.322,E2 -2959.322} C_VEL
LIN {X 0,Y 559.304,Z 438.605,A -85,B 0,C 180,E1 -2960.142,E2 -2960.142} C_VEL
LIN {X 0,Y 559.162,Z 447.113,A -85,B 0,C 180,E1 -2960.961,E2 -2960.961} C_VEL
LIN {X 0,Y 559.05,Z 454.961,A -85,B 0,C 180,E1 -2961.87,E2 -2961.87} C_VEL
LIN {X 0,Y 558.944,Z 462.623,A -85,B 0,C 180,E1 -2962.958,E2 -2962.958} C_VEL
LIN {X 0,Y 558.935,Z 469.68,A -85,B 0,C 180,E1 -2964.227,E2 -2964.227} C_VEL
LIN {X 0,Y 558.826,Z 474.373,A -85,B 0,C 180,E1 -2965.311,E2 -2965.311} C_VEL
LIN {X 0,Y 558.836,Z 477.958,A -85,B 0,C 180,E1 -2966.395,E2 -2966.395} C_VEL
LIN {X 0,Y 558.799,Z 479.807,A -85,B 0,C 180,E1 -2967.116,E2 -2967.116} C_VEL
LIN {X 0,Y 558.745,Z 482.183,A -85,B 0,C 180,E1 -2968.559,E2 -2968.559} C_VEL
LIN {X 0,Y 558.74,Z 483,A -85,B 0,C 180,E1 -2970,E2 -2970} C_VEL
LIN {X 0,Y 558.745,Z 482.185,A -85,B 0,C 180,E1 -2971.442,E2 -2971.442} C_VEL
LIN {X 0,Y 558.799,Z 479.81,A -85,B 0,C 180,E1 -2972.884,E2 -2972.884} C_VEL
LIN {X 0,Y 558.844,Z 476.895,A -85,B 0,C 180,E1 -2973.966,E2 -2973.966} C_VEL
LIN {X 0,Y 558.798,Z 472.948,A -85,B 0,C 180,E1 -2975.051,E2 -2975.051} C_VEL
LIN {X 0,Y 558.919,Z 467.867,A -85,B 0,C 180,E1 -2976.136,E2 -2976.136} C_VEL
LIN {X 0,Y 558.977,Z 461.467,A -85,B 0,C 180,E1 -2977.223,E2 -2977.223} C_VEL
LIN {X 0,Y 559.099,Z 453.477,A -85,B 0,C 180,E1 -2978.312,E2 -2978.312} C_VEL
LIN {X 0,Y 559.185,Z 445.333,A -85,B 0,C 180,E1 -2979.221,E2 -2979.221} C_VEL
LIN {X 0,Y 559.355,Z 435.398,A -85,B 0,C 180,E1 -2980.131,E2 -2980.131} C_VEL
LIN {X 0,Y 559.534,Z 424.403,A -85,B 0,C 180,E1 -2980.937,E2 -2980.937} C_VEL
LIN {X 0,Y 559.672,Z 412.457,A -85,B 0,C 180,E1 -2981.628,E2 -2981.628} C_VEL
LIN {X 0,Y 559.81,Z 399.767,A -85,B 0,C 180,E1 -2982.185,E2 -2982.185} C_VEL
LIN {X 0,Y 559.972,Z 386.343,A -85,B 0,C 180,E1 -2982.596,E2 -2982.596} C_VEL
LIN {X 0,Y 560.051,Z 373.082,A -85,B 0,C 180,E1 -2982.847,E2 -2982.847} C_VEL
LIN {X 0,Y 560.211,Z 276.506,A -85,B 0,C 180,E1 -2984.091,E2 -2984.091} C_VEL
LIN {X 0,Y 559.395,Z 270.792,A -85,B 0,C 180,E1 -2984.204,E2 -2984.204} C_VEL
LIN {X 0,Y 559.607,Z 248.085,A -85,B 0,C 180,E1 -2987.542,E2 -2987.542} C_VEL
LIN {X 0,Y 559.923,Z 227.677,A -85,B 0,C 180,E1 -2990.576,E2 -2990.576} C_VEL
LIN {X 0,Y 560.026,Z 214.897,A -85,B 0,C 180,E1 -2992.505,E2 -2992.505} C_VEL
LIN {X 0,Y 559.128,Z 209.842,A -85,B 0,C 180,E1 -2993.343,E2 -2993.343} C_VEL
LIN {X 0,Y 559.162,Z 209.831,A -85,B 0,C 180,E1 -2996.098,E2 -2996.098} C_VEL
LIN {X 0,Y 559.14,Z 209.832,A -85,B 0,C 180,E1 -2998.531,E2 -2998.531} C_VEL
LIN {X 0,Y 559.143,Z 209.838,A -85,B 0,C 180,E1 -3001.272,E2 -3001.272} C_VEL
LIN {X 0,Y 559.167,Z 209.83,A -85,B 0,C 180,E1 -3003.949,E2 -3003.949} C_VEL
LIN {X 0,Y 559.132,Z 209.836,A -85,B 0,C 180,E1 -3007.109,E2 -3007.109} C_VEL
LIN {X 0,Y 559.16,Z 209.831,A -85,B 0,C 180,E1 -3009.941,E2 -3009.941} C_VEL
LIN {X 0,Y 559.154,Z 209.83,A -85,B 0,C 180,E1 -3012.744,E2 -3012.744} C_VEL
LIN {X 0,Y 559.127,Z 209.839,A -85,B 0,C 180,E1 -3015.259,E2 -3015.259} C_VEL
LIN {X 0,Y 559.162,Z 209.828,A -85,B 0,C 180,E1 -3018.229,E2 -3018.229} C_VEL
LIN {X 0,Y 559.173,Z 209.832,A -85,B 0,C 180,E1 -3021.192,E2 -3021.192} C_VEL
LIN {X 0,Y 559.119,Z 209.838,A -85,B 0,C 180,E1 -3023.788,E2 -3023.788} C_VEL
LIN {X 0,Y 559.149,Z 209.828,A -85,B 0,C 180,E1 -3026.424,E2 -3026.424} C_VEL
LIN {X 0,Y 559.154,Z 209.831,A -85,B 0,C 180,E1 -3028.981,E2 -3028.981} C_VEL
LIN {X 0,Y 559.135,Z 209.838,A -85,B 0,C 180,E1 -3031.625,E2 -3031.625} C_VEL
LIN {X 0,Y 559.17,Z 209.828,A -85,B 0,C 180,E1 -3033.902,E2 -3033.902} C_VEL
LIN {X 0,Y 559.139,Z 209.831,A -85,B 0,C 180,E1 -3036.572,E2 -3036.572} C_VEL
LIN {X 0,Y 559.177,Z 209.834,A -85,B 0,C 180,E1 -3039.395,E2 -3039.395} C_VEL
LIN {X 0,Y 559.137,Z 209.836,A -85,B 0,C 180,E1 -3041.685,E2 -3041.685} C_VEL
LIN {X 0,Y 559.16,Z 209.83,A -85,B 0,C 180,E1 -3043.948,E2 -3043.948} C_VEL
LIN {X 0,Y 559.169,Z 209.827,A -85,B 0,C 180,E1 -3046.184,E2 -3046.184} C_VEL
LIN {X 0,Y 559.195,Z 209.827,A -85,B 0,C 180,E1 -3049.134,E2 -3049.134} C_VEL
LIN {X 0,Y 559.199,Z 209.823,A -85,B 0,C 180,E1 -3052.054,E2 -3052.054} C_VEL
LIN {X 0,Y 559.25,Z 209.819,A -85,B 0,C 180,E1 -3054.953,E2 -3054.953} C_VEL
LIN {X 0,Y 559.255,Z 209.818,A -85,B 0,C 180,E1 -3057.839,E2 -3057.839} C_VEL
LIN {X 0,Y 559.263,Z 209.816,A -85,B 0,C 180,E1 -3060.72,E2 -3060.72} C_VEL
LIN {X 0,Y 559.229,Z 209.82,A -85,B 0,C 180,E1 -3062.882,E2 -3062.882} C_VEL
LIN {X 0,Y 559.229,Z 209.824,A -85,B 0,C 180,E1 -3065.77,E2 -3065.77} C_VEL
LIN {X 0,Y 559.168,Z 209.826,A -85,B 0,C 180,E1 -3068.675,E2 -3068.675} C_VEL
LIN {X 0,Y 559.206,Z 209.829,A -85,B 0,C 180,E1 -3071.601,E2 -3071.601} C_VEL
LIN {X 0,Y 559.182,Z 209.825,A -85,B 0,C 180,E1 -3074.588,E2 -3074.588} C_VEL
LIN {X 0,Y 559.137,Z 209.837,A -85,B 0,C 180,E1 -3077.558,E2 -3077.558} C_VEL
LIN {X 0,Y 559.166,Z 209.83,A -85,B 0,C 180,E1 -3079.838,E2 -3079.838} C_VEL
LIN {X 0,Y 559.137,Z 209.83,A -85,B 0,C 180,E1 -3082.153,E2 -3082.153} C_VEL
LIN {X 0,Y 559.143,Z 209.836,A -85,B 0,C 180,E1 -3085.179,E2 -3085.179} C_VEL
LIN {X 0,Y 559.138,Z 209.836,A -85,B 0,C 180,E1 -3087.715,E2 -3087.715} C_VEL
LIN {X 0,Y 559.136,Z 209.83,A -85,B 0,C 180,E1 -3090.591,E2 -3090.591} C_VEL
LIN {X 0,Y 558.474,Z 209.921,A -85,B 0,C 180,E1 -3091.193,E2 -3091.193} C_VEL
LIN {X 0,Y 555.614,Z 210.273,A -85,B 0,C 180,E1 -3092.169,E2 -3092.169} C_VEL
LIN {X 0,Y 553.204,Z 210.573,A -85,B 0,C 180,E1 -3092.955,E2 -3092.955} C_VEL
LIN {X 0,Y 552.184,Z 210.704,A -85,B 0,C 180,E1 -3093.561,E2 -3093.561} C_VEL
LIN {X 0,Y 552.109,Z 210.707,A -85,B 0,C 180,E1 -3093.767,E2 -3093.767} C_VEL
LIN {X 0,Y 552.1,Z 210.708,A -85,B 0,C 180,E1 -3096.748,E2 -3096.748} C_VEL
LIN {X 0,Y 552.13,Z 210.712,A -85,B 0,C 180,E1 -3099.528,E2 -3099.528} C_VEL
LIN {X 0,Y 552.111,Z 210.706,A -85,B 0,C 180,E1 -3102.428,E2 -3102.428} C_VEL
LIN {X 0,Y 552.077,Z 210.717,A -85,B 0,C 180,E1 -3105.561,E2 -3105.561} C_VEL
LIN {X 0,Y 552.123,Z 210.707,A -85,B 0,C 180,E1 -3108.679,E2 -3108.679} C_VEL
LIN {X 0,Y 552.118,Z 210.716,A -85,B 0,C 180,E1 -3111.411,E2 -3111.411} C_VEL
LIN {X 0,Y 552.077,Z 210.712,A -85,B 0,C 180,E1 -3114.156,E2 -3114.156} C_VEL
LIN {X 0,Y 552.11,Z 210.709,A -85,B 0,C 180,E1 -3116.814,E2 -3116.814} C_VEL
LIN {X 0,Y 552.104,Z 210.715,A -85,B 0,C 180,E1 -3119.391,E2 -3119.391} C_VEL
LIN {X 0,Y 552.081,Z 210.714,A -85,B 0,C 180,E1 -3121.9,E2 -3121.9} C_VEL
LIN {X 0,Y 552.131,Z 210.718,A -85,B 0,C 180,E1 -3124.052,E2 -3124.052} C_VEL
LIN {X 0,Y 552.54,Z 215.285,A -85,B 0,C 180,E1 -3124.879,E2 -3124.879} C_VEL
LIN {X 0,Y 552.336,Z 231.506,A -85,B 0,C 180,E1 -3127.757,E2 -3127.757} C_VEL
LIN {X 0,Y 552.209,Z 242.287,A -85,B 0,C 180,E1 -3129.683,E2 -3129.683} C_VEL
LIN {X 0,Y 553.402,Z 250.34,A -85,B 0,C 180,E1 -3129.825,E2 -3129.825} C_VEL
LIN {X 0,Y 553.077,Z 349.768,A -85,B 0,C 180,E1 -3131.141,E2 -3131.141} C_VEL
LIN {X 0,Y 552.967,Z 363.054,A -85,B 0,C 180,E1 -3131.474,E2 -3131.474} C_VEL
LIN {X 0,Y 552.81,Z 375.814,A -85,B 0,C 180,E1 -3131.948,E2 -3131.948} C_VEL
LIN {X 0,Y 552.658,Z 387.538,A -85,B 0,C 180,E1 -3132.542,E2 -3132.542} C_VEL
LIN {X 0,Y 552.448,Z 398.798,A -85,B 0,C 180,E1 -3133.272,E2 -3133.272} C_VEL
LIN {X 0,Y 552.26,Z 409.3,A -85,B 0,C 180,E1 -3134.121,E2 -3134.121} C_VEL
LIN {X 0,Y 552.104,Z 418.681,A -85,B 0,C 180,E1 -3135.062,E2 -3135.062} C_VEL
LIN {X 0,Y 551.975,Z 427.762,A -85,B 0,C 180,E1 -3136.188,E2 -3136.188} C_VEL
LIN {X 0,Y 551.887,Z 435.023,A -85,B 0,C 180,E1 -3137.31,E2 -3137.31} C_VEL
LIN {X 0,Y 551.775,Z 441.491,A -85,B 0,C 180,E1 -3138.592,E2 -3138.592} C_VEL
LIN {X 0,Y 551.724,Z 445.899,A -85,B 0,C 180,E1 -3139.727,E2 -3139.727} C_VEL
LIN {X 0,Y 551.715,Z 448.177,A -85,B 0,C 180,E1 -3140.468,E2 -3140.468} C_VEL
LIN {X 0,Y 551.686,Z 449.98,A -85,B 0,C 180,E1 -3141.207,E2 -3141.207} C_VEL
LIN {X 0,Y 551.699,Z 451.334,A -85,B 0,C 180,E1 -3141.945,E2 -3141.945} C_VEL
LIN {X 0,Y 551.747,Z 452.851,A -85,B 0,C 180,E1 -3143.417,E2 -3143.417} C_VEL
LIN {X 0,Y 551.708,Z 452.984,A -85,B 0,C 180,E1 -3144.151,E2 -3144.151} C_VEL
LIN {X 0,Y 551.698,Z 452.06,A -85,B 0,C 180,E1 -3145.616,E2 -3145.616} C_VEL
LIN {X 0,Y 551.732,Z 451.019,A -85,B 0,C 180,E1 -3146.348,E2 -3146.348} C_VEL
LIN {X 0,Y 551.721,Z 449.537,A -85,B 0,C 180,E1 -3147.079,E2 -3147.079} C_VEL
LIN {X 0,Y 551.74,Z 446.534,A -85,B 0,C 180,E1 -3148.175,E2 -3148.175} C_VEL
LIN {X 0,Y 551.715,Z 442.498,A -85,B 0,C 180,E1 -3149.27,E2 -3149.27} C_VEL
LIN {X 0,Y 551.864,Z 436.302,A -85,B 0,C 180,E1 -3150.547,E2 -3150.547} C_VEL
LIN {X 0,Y 551.935,Z 429.584,A -85,B 0,C 180,E1 -3151.642,E2 -3151.642} C_VEL
LIN {X 0,Y 552.041,Z 421.259,A -85,B 0,C 180,E1 -3152.736,E2 -3152.736} C_VEL
LIN {X 0,Y 552.157,Z 412.709,A -85,B 0,C 180,E1 -3153.649,E2 -3153.649} C_VEL
LIN {X 0,Y 552.388,Z 402.204,A -85,B 0,C 180,E1 -3154.561,E2 -3154.561} C_VEL
LIN {X 0,Y 552.562,Z 391.832,A -85,B 0,C 180,E1 -3155.291,E2 -3155.291} C_VEL
LIN {X 0,Y 552.72,Z 380.397,A -85,B 0,C 180,E1 -3155.93,E2 -3155.93} C_VEL
LIN {X 0,Y 552.929,Z 368.537,A -85,B 0,C 180,E1 -3156.431,E2 -3156.431} C_VEL
LIN {X 0,Y 553.074,Z 355.715,A -85,B 0,C 180,E1 -3156.819,E2 -3156.819} C_VEL
LIN {X 0,Y 553.143,Z 342.066,A -85,B 0,C 180,E1 -3157.07,E2 -3157.07} C_VEL
LIN {X 0,Y 553.327,Z 248.731,A -85,B 0,C 180,E1 -3158.288,E2 -3158.288} C_VEL
LIN {X 0,Y 552.255,Z 242.193,A -85,B 0,C 180,E1 -3158.418,E2 -3158.418} C_VEL
LIN {X 0,Y 552.457,Z 225.391,A -85,B 0,C 180,E1 -3161.431,E2 -3161.431} C_VEL
LIN {X 0,Y 552.515,Z 213.214,A -85,B 0,C 180,E1 -3163.61,E2 -3163.61} C_VEL
LIN {X 0,Y 552.165,Z 210.707,A -85,B 0,C 180,E1 -3164.078,E2 -3164.078} C_VEL
LIN {X 0,Y 552.12,Z 210.708,A -85,B 0,C 180,E1 -3167.314,E2 -3167.314} C_VEL
LIN {X 0,Y 552.13,Z 210.705,A -85,B 0,C 180,E1 -3170.101,E2 -3170.101} C_VEL
LIN {X 0,Y 552.095,Z 210.714,A -85,B 0,C 180,E1 -3172.451,E2 -3172.451} C_VEL
LIN {X 0,Y 552.14,Z 210.703,A -85,B 0,C 180,E1 -3175.346,E2 -3175.346} C_VEL
LIN {X 0,Y 552.081,Z 210.711,A -85,B 0,C 180,E1 -3178.1,E2 -3178.1} C_VEL
LIN {X 0,Y 552.104,Z 210.716,A -85,B 0,C 180,E1 -3180.609,E2 -3180.609} C_VEL
LIN {X 0,Y 552.115,Z 210.708,A -85,B 0,C 180,E1 -3183.186,E2 -3183.186} C_VEL
LIN {X 0,Y 552.078,Z 210.71,A -85,B 0,C 180,E1 -3185.844,E2 -3185.844} C_VEL
LIN {X 0,Y 552.118,Z 210.714,A -85,B 0,C 180,E1 -3188.589,E2 -3188.589} C_VEL
LIN {X 0,Y 552.122,Z 210.705,A -85,B 0,C 180,E1 -3191.446,E2 -3191.446} C_VEL
LIN {X 0,Y 552.093,Z 210.716,A -85,B 0,C 180,E1 -3194.531,E2 -3194.531} C_VEL
LIN {X 0,Y 552.111,Z 210.706,A -85,B 0,C 180,E1 -3197.587,E2 -3197.587} C_VEL
LIN {X 0,Y 552.13,Z 210.71,A -85,B 0,C 180,E1 -3200.473,E2 -3200.473} C_VEL
LIN {X 0,Y 552.1,Z 210.708,A -85,B 0,C 180,E1 -3203.318,E2 -3203.318} C_VEL
LIN {X 0,Y 552.127,Z 210.705,A -85,B 0,C 180,E1 -3205.939,E2 -3205.939} C_VEL
LIN {X 0,Y 552.121,Z 210.713,A -85,B 0,C 180,E1 -3208.54,E2 -3208.54} C_VEL
LIN {X 0,Y 552.106,Z 210.707,A -85,B 0,C 180,E1 -3211.442,E2 -3211.442} C_VEL
LIN {X 0,Y 552.106,Z 210.707,A -85,B 0,C 180,E1 -3213.542,E2 -3213.542} C_VEL
LIN {X 0,Y 552.097,Z 210.716,A -85,B 0,C 180,E1 -3216.758,E2 -3216.758} C_VEL
LIN {X 0,Y 552.118,Z 210.708,A -85,B 0,C 180,E1 -3219.12,E2 -3219.12} C_VEL
LIN {X 0,Y 552.095,Z 210.708,A -85,B 0,C 180,E1 -3221.443,E2 -3221.443} C_VEL
LIN {X 0,Y 552.109,Z 210.706,A -85,B 0,C 180,E1 -3223.737,E2 -3223.737} C_VEL
LIN {X 0,Y 552.131,Z 210.705,A -85,B 0,C 180,E1 -3226.004,E2 -3226.004} C_VEL
LIN {X 0,Y 552.162,Z 210.704,A -85,B 0,C 180,E1 -3228.993,E2 -3228.993} C_VEL
LIN {X 0,Y 552.15,Z 210.702,A -85,B 0,C 180,E1 -3231.951,E2 -3231.951} C_VEL
LIN {X 0,Y 552.223,Z 210.697,A -85,B 0,C 180,E1 -3234.889,E2 -3234.889} C_VEL
LIN {X 0,Y 552.224,Z 210.692,A -85,B 0,C 180,E1 -3237.812,E2 -3237.812} C_VEL
LIN {X 0,Y 552.242,Z 210.697,A -85,B 0,C 180,E1 -3240.729,E2 -3240.729} C_VEL
LIN {X 0,Y 552.202,Z 210.699,A -85,B 0,C 180,E1 -3242.918,E2 -3242.918} C_VEL
LIN {X 0,Y 552.193,Z 210.696,A -85,B 0,C 180,E1 -3245.844,E2 -3245.844} C_VEL
LIN {X 0,Y 552.152,Z 210.707,A -85,B 0,C 180,E1 -3248.786,E2 -3248.786} C_VEL
LIN {X 0,Y 552.163,Z 210.699,A -85,B 0,C 180,E1 -3251.75,E2 -3251.75} C_VEL
LIN {X 0,Y 552.137,Z 210.71,A -85,B 0,C 180,E1 -3254.748,E2 -3254.748} C_VEL
LIN {X 0,Y 552.097,Z 210.708,A -85,B 0,C 180,E1 -3257.789,E2 -3257.789} C_VEL
LIN {X 0,Y 552.127,Z 210.707,A -85,B 0,C 180,E1 -3260.101,E2 -3260.101} C_VEL
LIN {X 0,Y 552.091,Z 210.716,A -85,B 0,C 180,E1 -3262.451,E2 -3262.451} C_VEL
LIN {X 0,Y 552.138,Z 210.703,A -85,B 0,C 180,E1 -3265.346,E2 -3265.346} C_VEL
LIN {X 0,Y 552.078,Z 210.713,A -85,B 0,C 180,E1 -3268.1,E2 -3268.1} C_VEL
LIN {X 0,Y 552.102,Z 210.717,A -85,B 0,C 180,E1 -3270.609,E2 -3270.609} C_VEL
LIN {X 0,Y 552.108,Z 210.708,A -85,B 0,C 180,E1 -3273.186,E2 -3273.186} C_VEL
LIN {X 0,Y 552.075,Z 210.711,A -85,B 0,C 180,E1 -3275.845,E2 -3275.845} C_VEL
LIN {X 0,Y 552.116,Z 210.715,A -85,B 0,C 180,E1 -3278.589,E2 -3278.589} C_VEL
LIN {X 0,Y 552.12,Z 210.705,A -85,B 0,C 180,E1 -3281.446,E2 -3281.446} C_VEL
LIN {X 0,Y 552.076,Z 210.72,A -85,B 0,C 180,E1 -3284.53,E2 -3284.53} C_VEL
LIN {X 0,Y 552.11,Z 210.706,A -85,B 0,C 180,E1 -3287.587,E2 -3287.587} C_VEL
LIN {X 0,Y 552.129,Z 210.713,A -85,B 0,C 180,E1 -3290.473,E2 -3290.473} C_VEL
LIN {X 0,Y 552.1,Z 210.708,A -85,B 0,C 180,E1 -3293.318,E2 -3293.318} C_VEL
LIN {X 0,Y 552.127,Z 210.705,A -85,B 0,C 180,E1 -3295.939,E2 -3295.939} C_VEL
LIN {X 0,Y 552.121,Z 210.715,A -85,B 0,C 180,E1 -3298.541,E2 -3298.541} C_VEL
LIN {X 0,Y 552.105,Z 210.708,A -85,B 0,C 180,E1 -3301.442,E2 -3301.442} C_VEL
LIN {X 0,Y 552.105,Z 210.708,A -85,B 0,C 180,E1 -3303.543,E2 -3303.543} C_VEL
LIN {X 0,Y 552.124,Z 210.853,A -85,B 0,C 180,E1 -3306.551,E2 -3306.551} C_VEL
LIN {X 0,Y 553.118,Z 217.321,A -85,B 0,C 180,E1 -3307.593,E2 -3307.593} C_VEL
LIN {X 0,Y 552.855,Z 234.221,A -85,B 0,C 180,E1 -3310.17,E2 -3310.17} C_VEL
LIN {X 0,Y 552.544,Z 252.999,A -85,B 0,C 180,E1 -3312.99,E2 -3312.99} C_VEL
LIN {X 0,Y 552.366,Z 270.741,A -85,B 0,C 180,E1 -3315.625,E2 -3315.625} C_VEL
LIN {X 0,Y 553.416,Z 278.658,A -85,B 0,C 180,E1 -3315.763,E2 -3315.763} C_VEL
LIN {X 0,Y 553.117,Z 378.897,A -85,B 0,C 180,E1 -3317.082,E2 -3317.082} C_VEL
LIN {X 0,Y 552.982,Z 392.185,A -85,B 0,C 180,E1 -3317.406,E2 -3317.406} C_VEL
LIN {X 0,Y 552.84,Z 404.359,A -85,B 0,C 180,E1 -3317.845,E2 -3317.845} C_VEL
LIN {X 0,Y 552.659,Z 415.185,A -85,B 0,C 180,E1 -3318.366,E2 -3318.366} C_VEL
LIN {X 0,Y 552.541,Z 426.901,A -85,B 0,C 180,E1 -3319.094,E2 -3319.094} C_VEL
LIN {X 0,Y 552.295,Z 437.536,A -85,B 0,C 180,E1 -3319.923,E2 -3319.923} C_VEL
LIN {X 0,Y 552.126,Z 447.114,A -85,B 0,C 180,E1 -3320.845,E2 -3320.845} C_VEL
LIN {X 0,Y 552.013,Z 454.961,A -85,B 0,C 180,E1 -3321.765,E2 -3321.765} C_VEL
LIN {X 0,Y 551.889,Z 462.621,A -85,B 0,C 180,E1 -3322.868,E2 -3322.868} C_VEL
LIN {X 0,Y 551.867,Z 469.68,A -85,B 0,C 180,E1 -3324.153,E2 -3324.153} C_VEL
LIN {X 0,Y 551.725,Z 474.373,A -85,B 0,C 180,E1 -3325.251,E2 -3325.251} C_VEL
LIN {X 0,Y 551.75,Z 477.958,A -85,B 0,C 180,E1 -3326.348,E2 -3326.348} C_VEL
LIN {X 0,Y 551.723,Z 479.807,A -85,B 0,C 180,E1 -3327.079,E2 -3327.079} C_VEL
LIN {X 0,Y 551.645,Z 482.182,A -85,B 0,C 180,E1 -3328.54,E2 -3328.54} C_VEL
LIN {X 0,Y 551.64,Z 483,A -85,B 0,C 180,E1 -3330,E2 -3330} C_VEL
LIN {X 0,Y 551.645,Z 482.184,A -85,B 0,C 180,E1 -3331.46,E2 -3331.46} C_VEL
LIN {X 0,Y 551.723,Z 479.81,A -85,B 0,C 180,E1 -3332.921,E2 -3332.921} C_VEL
LIN {X 0,Y 551.764,Z 476.895,A -85,B 0,C 180,E1 -3334.017,E2 -3334.017} C_VEL
LIN {X 0,Y 551.723,Z 472.948,A -85,B 0,C 180,E1 -3335.116,E2 -3335.116} C_VEL
LIN {X 0,Y 551.801,Z 467.198,A -85,B 0,C 180,E1 -3336.34,E2 -3336.34} C_VEL
LIN {X 0,Y 551.926,Z 460.235,A -85,B 0,C 180,E1 -3337.5,E2 -3337.5} C_VEL
LIN {X 0,Y 552.082,Z 451.992,A -85,B 0,C 180,E1 -3338.602,E2 -3338.602} C_VEL
LIN {X 0,Y 552.224,Z 443.539,A -85,B 0,C 180,E1 -3339.523,E2 -3339.523} C_VEL
LIN {X 0,Y 552.425,Z 433.09,A -85,B 0,C 180,E1 -3340.445,E2 -3340.445} C_VEL
LIN {X 0,Y 552.605,Z 422.295,A -85,B 0,C 180,E1 -3341.213,E2 -3341.213} C_VEL
LIN {X 0,Y 552.751,Z 411.403,A -85,B 0,C 180,E1 -3341.831,E2 -3341.831} C_VEL
LIN {X 0,Y 552.871,Z 399.742,A -85,B 0,C 180,E1 -3342.34,E2 -3342.34} C_VEL
LIN {X 0,Y 553.044,Z 386.3,A -85,B 0,C 180,E1 -3342.756,E2 -3342.756} C_VEL
LIN {X 0,Y 553.145,Z 373.024,A -85,B 0,C 180,E1 -3343.01,E2 -3343.01} C_VEL
LIN {X 0,Y 553.358,Z 277.564,A -85,B 0,C 180,E1 -3344.253,E2 -3344.253} C_VEL
LIN {X 0,Y 552.359,Z 270.601,A -85,B 0,C 180,E1 -3344.394,E2 -3344.394} C_VEL
LIN {X 0,Y 552.633,Z 247.882,A -85,B 0,C 180,E1 -3347.771,E2 -3347.771} C_VEL
LIN {X 0,Y 552.969,Z 228.75,A -85,B 0,C 180,E1 -3350.652,E2 -3350.652} C_VEL
LIN {X 0,Y 553.055,Z 215.969,A -85,B 0,C 180,E1 -3352.607,E2 -3352.607} C_VEL
LIN {X 0,Y 552.098,Z 210.717,A -85,B 0,C 180,E1 -3353.493,E2 -3353.493} C_VEL
LIN {X 0,Y 552.105,Z 210.709,A -85,B 0,C 180,E1 -3356.457,E2 -3356.457} C_VEL
LIN {X 0,Y 552.099,Z 210.712,A -85,B 0,C 180,E1 -3358.929,E2 -3358.929} C_VEL
LIN {X 0,Y 552.113,Z 210.715,A -85,B 0,C 180,E1 -3361.475,E2 -3361.475} C_VEL
LIN {X 0,Y 552.133,Z 210.705,A -85,B 0,C 180,E1 -3364.17,E2 -3364.17} C_VEL
LIN {X 0,Y 552.1,Z 210.709,A -85,B 0,C 180,E1 -3366.748,E2 -3366.748} C_VEL
LIN {X 0,Y 552.129,Z 210.713,A -85,B 0,C 180,E1 -3369.527,E2 -3369.527} C_VEL
LIN {X 0,Y 552.11,Z 210.707,A -85,B 0,C 180,E1 -3372.427,E2 -3372.427} C_VEL
LIN {X 0,Y 552.077,Z 210.719,A -85,B 0,C 180,E1 -3375.56,E2 -3375.56} C_VEL
LIN {X 0,Y 552.121,Z 210.705,A -85,B 0,C 180,E1 -3378.679,E2 -3378.679} C_VEL
LIN {X 0,Y 552.115,Z 210.715,A -85,B 0,C 180,E1 -3381.411,E2 -3381.411} C_VEL
LIN {X 0,Y 552.072,Z 210.712,A -85,B 0,C 180,E1 -3384.155,E2 -3384.155} C_VEL
LIN {X 0,Y 552.108,Z 210.706,A -85,B 0,C 180,E1 -3386.814,E2 -3386.814} C_VEL
LIN {X 0,Y 552.102,Z 210.716,A -85,B 0,C 180,E1 -3389.391,E2 -3389.391} C_VEL
LIN {X 0,Y 552.078,Z 210.713,A -85,B 0,C 180,E1 -3391.9,E2 -3391.9} C_VEL
LIN {X 0,Y 552.138,Z 210.702,A -85,B 0,C 180,E1 -3394.654,E2 -3394.654} C_VEL
LIN {X 0,Y 552.092,Z 210.716,A -85,B 0,C 180,E1 -3397.549,E2 -3397.549} C_VEL
LIN {X 0,Y 552.146,Z 210.702,A -85,B 0,C 180,E1 -3400.375,E2 -3400.375} C_VEL
LIN {X 0,Y 552.133,Z 210.706,A -85,B 0,C 180,E1 -3402.977,E2 -3402.977} C_VEL
LIN {X 0,Y 552.134,Z 210.705,A -85,B 0,C 180,E1 -3406.004,E2 -3406.004} C_VEL
LIN {X 0,Y 552.163,Z 210.701,A -85,B 0,C 180,E1 -3408.993,E2 -3408.993} C_VEL
LIN {X 0,Y 552.155,Z 210.702,A -85,B 0,C 180,E1 -3411.952,E2 -3411.952} C_VEL
LIN {X 0,Y 552.224,Z 210.693,A -85,B 0,C 180,E1 -3414.889,E2 -3414.889} C_VEL
LIN {X 0,Y 552.226,Z 210.694,A -85,B 0,C 180,E1 -3417.812,E2 -3417.812} C_VEL
LIN {X 0,Y 552.234,Z 210.691,A -85,B 0,C 180,E1 -3420.729,E2 -3420.729} C_VEL
LIN {X 0,Y 552.196,Z 210.697,A -85,B 0,C 180,E1 -3422.918,E2 -3422.918} C_VEL
LIN {X 0,Y 552.198,Z 210.699,A -85,B 0,C 180,E1 -3425.844,E2 -3425.844} C_VEL
LIN {X 0,Y 552.139,Z 210.702,A -85,B 0,C 180,E1 -3428.786,E2 -3428.786} C_VEL
LIN {X 0,Y 552.163,Z 210.703,A -85,B 0,C 180,E1 -3431.751,E2 -3431.751} C_VEL
LIN {X 0,Y 552.13,Z 210.704,A -85,B 0,C 180,E1 -3434.749,E2 -3434.749} C_VEL
LIN {X 0,Y 552.095,Z 210.71,A -85,B 0,C 180,E1 -3437.789,E2 -3437.789} C_VEL
LIN {X 0,Y 552.126,Z 210.705,A -85,B 0,C 180,E1 -3440.102,E2 -3440.102} C_VEL
LIN {X 0,Y 552.089,Z 210.707,A -85,B 0,C 180,E1 -3442.451,E2 -3442.451} C_VEL
LIN {X 0,Y 552.088,Z 210.718,A -85,B 0,C 180,E1 -3445.335,E2 -3445.335} C_VEL
LIN {X 0,Y 552.089,Z 210.71,A -85,B 0,C 180,E1 -3448.1,E2 -3448.1} C_VEL
LIN {X 0,Y 552.099,Z 210.707,A -85,B 0,C 180,E1 -3450.61,E2 -3450.61} C_VEL
LIN {X 0,Y 552.117,Z 210.712,A -85,B 0,C 180,E1 -3453.186,E2 -3453.186} C_VEL
LIN {X 0,Y 552.109,Z 210.707,A -85,B 0,C 180,E1 -3453.767,E2 -3453.767} C_VEL
LIN {X 0,Y 551.473,Z 210.789,A -85,B 0,C 180,E1 -3454.375,E2 -3454.375} C_VEL
LIN {X 0,Y 548.651,Z 211.147,A -85,B 0,C 180,E1 -3455.363,E2 -3455.363} C_VEL
LIN {X 0,Y 546.231,Z 211.442,A -85,B 0,C 180,E1 -3456.158,E2 -3456.158} C_VEL
LIN {X 0,Y 545.162,Z 211.573,A -85,B 0,C 180,E1 -3456.772,E2 -3456.772} C_VEL
LIN {X 0,Y 545.06,Z 211.587,A -85,B 0,C 180,E1 -3456.98,E2 -3456.98} C_VEL
LIN {X 0,Y 545.066,Z 211.585,A -85,B 0,C 180,E1 -3460.143,E2 -3460.143} C_VEL
LIN {X 0,Y 545.05,Z 211.587,A -85,B 0,C 180,E1 -3462.695,E2 -3462.695} C_VEL
LIN {X 0,Y 545.027,Z 211.595,A -85,B 0,C 180,E1 -3465.171,E2 -3465.171} C_VEL
LIN {X 0,Y 545.079,Z 211.584,A -85,B 0,C 180,E1 -3468.403,E2 -3468.403} C_VEL
LIN {X 0,Y 545.081,Z 211.584,A -85,B 0,C 180,E1 -3470.818,E2 -3470.818} C_VEL
LIN {X 0,Y 545.037,Z 211.595,A -85,B 0,C 180,E1 -3473.619,E2 -3473.619} C_VEL
LIN {X 0,Y 545.053,Z 211.586,A -85,B 0,C 180,E1 -3476.327,E2 -3476.327} C_VEL
LIN {X 0,Y 545.069,Z 211.587,A -85,B 0,C 180,E1 -3478.952,E2 -3478.952} C_VEL
LIN {X 0,Y 545.079,Z 211.589,A -85,B 0,C 180,E1 -3481.506,E2 -3481.506} C_VEL
LIN {X 0,Y 545.111,Z 211.69,A -85,B 0,C 180,E1 -3483.975,E2 -3483.975} C_VEL
LIN {X 0,Y 545.531,Z 216.418,A -85,B 0,C 180,E1 -3484.841,E2 -3484.841} C_VEL
LIN {X 0,Y 545.346,Z 232.162,A -85,B 0,C 180,E1 -3487.656,E2 -3487.656} C_VEL
LIN {X 0,Y 545.22,Z 242.392,A -85,B 0,C 180,E1 -3489.485,E2 -3489.485} C_VEL
LIN {X 0,Y 546.532,Z 250.56,A -85,B 0,C 180,E1 -3489.643,E2 -3489.643} C_VEL
LIN {X 0,Y 546.166,Z 349.545,A -85,B 0,C 180,E1 -3490.967,E2 -3490.967} C_VEL
LIN {X 0,Y 546.038,Z 362.967,A -85,B 0,C 180,E1 -3491.303,E2 -3491.303} C_VEL
LIN {X 0,Y 545.886,Z 375.25,A -85,B 0,C 180,E1 -3491.759,E2 -3491.759} C_VEL
LIN {X 0,Y 545.747,Z 387.088,A -85,B 0,C 180,E1 -3492.356,E2 -3492.356} C_VEL
LIN {X 0,Y 545.474,Z 397.886,A -85,B 0,C 180,E1 -3493.052,E2 -3493.052} C_VEL
LIN {X 0,Y 545.296,Z 408.571,A -85,B 0,C 180,E1 -3493.913,E2 -3493.913} C_VEL
LIN {X 0,Y 545.123,Z 418.13,A -85,B 0,C 180,E1 -3494.866,E2 -3494.866} C_VEL
LIN {X 0,Y 544.931,Z 427.285,A -85,B 0,C 180,E1 -3496.006,E2 -3496.006} C_VEL
LIN {X 0,Y 544.806,Z 434.626,A -85,B 0,C 180,E1 -3497.143,E2 -3497.143} C_VEL
LIN {X 0,Y 544.735,Z 439.557,A -85,B 0,C 180,E1 -3498.087,E2 -3498.087} C_VEL
LIN {X 0,Y 544.684,Z 444.323,A -85,B 0,C 180,E1 -3499.217,E2 -3499.217} C_VEL
LIN {X 0,Y 544.644,Z 447.952,A -85,B 0,C 180,E1 -3500.343,E2 -3500.343} C_VEL
LIN {X 0,Y 544.586,Z 449.821,A -85,B 0,C 180,E1 -3501.091,E2 -3501.091} C_VEL
LIN {X 0,Y 544.616,Z 451.215,A -85,B 0,C 180,E1 -3501.839,E2 -3501.839} C_VEL
LIN {X 0,Y 544.651,Z 452.802,A -85,B 0,C 180,E1 -3503.331,E2 -3503.331} C_VEL
LIN {X 0,Y 544.611,Z 452.998,A -85,B 0,C 180,E1 -3504.074,E2 -3504.074} C_VEL
LIN {X 0,Y 544.594,Z 452.143,A -85,B 0,C 180,E1 -3505.559,E2 -3505.559} C_VEL
LIN {X 0,Y 544.646,Z 451.136,A -85,B 0,C 180,E1 -3506.301,E2 -3506.301} C_VEL
LIN {X 0,Y 544.647,Z 449.722,A -85,B 0,C 180,E1 -3507.041,E2 -3507.041} C_VEL
LIN {X 0,Y 544.592,Z 445.571,A -85,B 0,C 180,E1 -3508.521,E2 -3508.521} C_VEL
LIN {X 0,Y 544.694,Z 441.261,A -85,B 0,C 180,E1 -3509.63,E2 -3509.63} C_VEL
LIN {X 0,Y 544.742,Z 435.789,A -85,B 0,C 180,E1 -3510.739,E2 -3510.739} C_VEL
LIN {X 0,Y 544.907,Z 428.969,A -85,B 0,C 180,E1 -3511.848,E2 -3511.848} C_VEL
LIN {X 0,Y 544.964,Z 420.465,A -85,B 0,C 180,E1 -3512.957,E2 -3512.957} C_VEL
LIN {X 0,Y 545.211,Z 411.749,A -85,B 0,C 180,E1 -3513.88,E2 -3513.88} C_VEL
LIN {X 0,Y 545.45,Z 401.05,A -85,B 0,C 180,E1 -3514.804,E2 -3514.804} C_VEL
LIN {X 0,Y 545.659,Z 390.303,A -85,B 0,C 180,E1 -3515.543,E2 -3515.543} C_VEL
LIN {X 0,Y 545.837,Z 378.306,A -85,B 0,C 180,E1 -3516.19,E2 -3516.19} C_VEL
LIN {X 0,Y 546.018,Z 365.754,A -85,B 0,C 180,E1 -3516.699,E2 -3516.699} C_VEL
LIN {X 0,Y 546.194,Z 353.31,A -85,B 0,C 180,E1 -3517.045,E2 -3517.045} C_VEL
LIN {X 0,Y 546.264,Z 335.815,A -85,B 0,C 180,E1 -3517.322,E2 -3517.322} C_VEL
LIN {X 0,Y 546.431,Z 249.397,A -85,B 0,C 180,E1 -3518.465,E2 -3518.465} C_VEL
LIN {X 0,Y 545.263,Z 242.453,A -85,B 0,C 180,E1 -3518.594,E2 -3518.594} C_VEL
LIN {X 0,Y 545.462,Z 225.219,A -85,B 0,C 180,E1 -3521.699,E2 -3521.699} C_VEL
LIN {X 0,Y 545.551,Z 214.667,A -85,B 0,C 180,E1 -3523.598,E2 -3523.598} C_VEL
LIN {X 0,Y 545.132,Z 211.584,A -85,B 0,C 180,E1 -3524.179,E2 -3524.179} C_VEL
LIN {X 0,Y 545.08,Z 211.584,A -85,B 0,C 180,E1 -3527.422,E2 -3527.422} C_VEL
LIN {X 0,Y 545.096,Z 211.584,A -85,B 0,C 180,E1 -3530.372,E2 -3530.372} C_VEL
LIN {X 0,Y 545.082,Z 211.582,A -85,B 0,C 180,E1 -3533.559,E2 -3533.559} C_VEL
LIN {X 0,Y 545.077,Z 211.583,A -85,B 0,C 180,E1 -3536.001,E2 -3536.001} C_VEL
LIN {X 0,Y 545.072,Z 211.592,A -85,B 0,C 180,E1 -3538.744,E2 -3538.744} C_VEL
LIN {X 0,Y 545.061,Z 211.584,A -85,B 0,C 180,E1 -3541.679,E2 -3541.679} C_VEL
LIN {X 0,Y 545.064,Z 211.592,A -85,B 0,C 180,E1 -3544.564,E2 -3544.564} C_VEL
LIN {X 0,Y 545.034,Z 211.589,A -85,B 0,C 180,E1 -3547.304,E2 -3547.304} C_VEL
LIN {X 0,Y 545.067,Z 211.586,A -85,B 0,C 180,E1 -3550.143,E2 -3550.143} C_VEL
LIN {X 0,Y 545.081,Z 211.585,A -85,B 0,C 180,E1 -3553.106,E2 -3553.106} C_VEL
LIN {X 0,Y 545.051,Z 211.589,A -85,B 0,C 180,E1 -3556.226,E2 -3556.226} C_VEL
LIN {X 0,Y 545.082,Z 211.588,A -85,B 0,C 180,E1 -3558.885,E2 -3558.885} C_VEL
LIN {X 0,Y 545.08,Z 211.589,A -85,B 0,C 180,E1 -3560.818,E2 -3560.818} C_VEL
LIN {X 0,Y 545.036,Z 211.587,A -85,B 0,C 180,E1 -3563.619,E2 -3563.619} C_VEL
LIN {X 0,Y 545.067,Z 211.588,A -85,B 0,C 180,E1 -3566.328,E2 -3566.328} C_VEL
LIN {X 0,Y 545.067,Z 211.588,A -85,B 0,C 180,E1 -3568.952,E2 -3568.952} C_VEL
LIN {X 0,Y 545.084,Z 211.581,A -85,B 0,C 180,E1 -3571.506,E2 -3571.506} C_VEL
LIN {X 0,Y 545.063,Z 211.585,A -85,B 0,C 180,E1 -3573.998,E2 -3573.998} C_VEL
LIN {X 0,Y 545.037,Z 211.589,A -85,B 0,C 180,E1 -3577.242,E2 -3577.242} C_VEL
LIN {X 0,Y 545.117,Z 211.583,A -85,B 0,C 180,E1 -3580.415,E2 -3580.415} C_VEL
LIN {X 0,Y 545.061,Z 211.584,A -85,B 0,C 180,E1 -3583.521,E2 -3583.521} C_VEL
LIN {X 0,Y 545.085,Z 211.581,A -85,B 0,C 180,E1 -3585.82,E2 -3585.82} C_VEL
LIN {X 0,Y 545.118,Z 211.583,A -85,B 0,C 180,E1 -3588.849,E2 -3588.849} C_VEL
LIN {X 0,Y 545.098,Z 211.58,A -85,B 0,C 180,E1 -3591.846,E2 -3591.846} C_VEL
LIN {X 0,Y 545.199,Z 211.573,A -85,B 0,C 180,E1 -3594.823,E2 -3594.823} C_VEL
LIN {X 0,Y 545.195,Z 211.568,A -85,B 0,C 180,E1 -3597.784,E2 -3597.784} C_VEL
LIN {X 0,Y 545.212,Z 211.573,A -85,B 0,C 180,E1 -3600.739,E2 -3600.739} C_VEL
LIN {X 0,Y 545.168,Z 211.575,A -85,B 0,C 180,E1 -3602.956,E2 -3602.956} C_VEL
LIN {X 0,Y 545.166,Z 211.572,A -85,B 0,C 180,E1 -3605.92,E2 -3605.92} C_VEL
LIN {X 0,Y 545.109,Z 211.583,A -85,B 0,C 180,E1 -3608.9,E2 -3608.9} C_VEL
LIN {X 0,Y 545.107,Z 211.579,A -85,B 0,C 180,E1 -3611.905,E2 -3611.905} C_VEL
LIN {X 0,Y 545.086,Z 211.585,A -85,B 0,C 180,E1 -3614.944,E2 -3614.944} C_VEL
LIN {X 0,Y 545.069,Z 211.585,A -85,B 0,C 180,E1 -3618.026,E2 -3618.026} C_VEL
LIN {X 0,Y 545.093,Z 211.587,A -85,B 0,C 180,E1 -3620.372,E2 -3620.372} C_VEL
LIN {X 0,Y 545.079,Z 211.582,A -85,B 0,C 180,E1 -3623.559,E2 -3623.559} C_VEL
LIN {X 0,Y 545.074,Z 211.584,A -85,B 0,C 180,E1 -3626.001,E2 -3626.001} C_VEL
LIN {X 0,Y 545.069,Z 211.59,A -85,B 0,C 180,E1 -3628.744,E2 -3628.744} C_VEL
LIN {X 0,Y 545.058,Z 211.584,A -85,B 0,C 180,E1 -3631.679,E2 -3631.679} C_VEL
LIN {X 0,Y 545.059,Z 211.594,A -85,B 0,C 180,E1 -3634.565,E2 -3634.565} C_VEL
LIN {X 0,Y 545.031,Z 211.588,A -85,B 0,C 180,E1 -3637.305,E2 -3637.305} C_VEL
LIN {X 0,Y 545.065,Z 211.587,A -85,B 0,C 180,E1 -3640.143,E2 -3640.143} C_VEL
LIN {X 0,Y 545.039,Z 211.594,A -85,B 0,C 180,E1 -3642.694,E2 -3642.694} C_VEL
LIN {X 0,Y 545.03,Z 211.589,A -85,B 0,C 180,E1 -3645.171,E2 -3645.171} C_VEL
LIN {X 0,Y 545.065,Z 211.585,A -85,B 0,C 180,E1 -3647.896,E2 -3647.896} C_VEL
LIN {X 0,Y 545.079,Z 211.587,A -85,B 0,C 180,E1 -3650.818,E2 -3650.818} C_VEL
LIN {X 0,Y 545.035,Z 211.587,A -85,B 0,C 180,E1 -3653.619,E2 -3653.619} C_VEL
LIN {X 0,Y 545.066,Z 211.59,A -85,B 0,C 180,E1 -3656.328,E2 -3656.328} C_VEL
LIN {X 0,Y 545.066,Z 211.587,A -85,B 0,C 180,E1 -3658.952,E2 -3658.952} C_VEL
LIN {X 0,Y 545.084,Z 211.583,A -85,B 0,C 180,E1 -3661.507,E2 -3661.507} C_VEL
LIN {X 0,Y 545.063,Z 211.588,A -85,B 0,C 180,E1 -3663.999,E2 -3663.999} C_VEL
LIN {X 0,Y 545.082,Z 211.744,A -85,B 0,C 180,E1 -3666.4,E2 -3666.4} C_VEL
LIN {X 0,Y 546.159,Z 218.301,A -85,B 0,C 180,E1 -3667.474,E2 -3667.474} C_VEL
LIN {X 0,Y 545.865,Z 235.567,A -85,B 0,C 180,E1 -3670.142,E2 -3670.142} C_VEL
LIN {X 0,Y 545.521,Z 254.074,A -85,B 0,C 180,E1 -3672.957,E2 -3672.957} C_VEL
LIN {X 0,Y 545.359,Z 270.762,A -85,B 0,C 180,E1 -3675.446,E2 -3675.446} C_VEL
LIN {X 0,Y 546.538,Z 278.921,A -85,B 0,C 180,E1 -3675.586,E2 -3675.586} C_VEL
LIN {X 0,Y 546.216,Z 378.692,A -85,B 0,C 180,E1 -3676.916,E2 -3676.916} C_VEL
LIN {X 0,Y 546.054,Z 391.983,A -85,B 0,C 180,E1 -3677.243,E2 -3677.243} C_VEL
LIN {X 0,Y 545.885,Z 404.158,A -85,B 0,C 180,E1 -3677.688,E2 -3677.688} C_VEL
LIN {X 0,Y 545.684,Z 415.227,A -85,B 0,C 180,E1 -3678.228,E2 -3678.228} C_VEL
LIN {X 0,Y 545.539,Z 426.753,A -85,B 0,C 180,E1 -3678.952,E2 -3678.952} C_VEL
LIN {X 0,Y 545.287,Z 437.423,A -85,B 0,C 180,E1 -3679.792,E2 -3679.792} C_VEL
LIN {X 0,Y 545.085,Z 447.038,A -85,B 0,C 180,E1 -3680.725,E2 -3680.725} C_VEL
LIN {X 0,Y 544.978,Z 454.921,A -85,B 0,C 180,E1 -3681.658,E2 -3681.658} C_VEL
LIN {X 0,Y 544.824,Z 462.617,A -85,B 0,C 180,E1 -3682.775,E2 -3682.775} C_VEL
LIN {X 0,Y 544.776,Z 469.679,A -85,B 0,C 180,E1 -3684.076,E2 -3684.076} C_VEL
LIN {X 0,Y 544.628,Z 474.373,A -85,B 0,C 180,E1 -3685.189,E2 -3685.189} C_VEL
LIN {X 0,Y 544.669,Z 477.958,A -85,B 0,C 180,E1 -3686.301,E2 -3686.301} C_VEL
LIN {X 0,Y 544.65,Z 479.807,A -85,B 0,C 180,E1 -3687.041,E2 -3687.041} C_VEL
LIN {X 0,Y 544.546,Z 482.182,A -85,B 0,C 180,E1 -3688.521,E2 -3688.521} C_VEL
LIN {X 0,Y 544.541,Z 483,A -85,B 0,C 180,E1 -3690,E2 -3690} C_VEL
LIN {X 0,Y 544.546,Z 482.183,A -85,B 0,C 180,E1 -3691.479,E2 -3691.479} C_VEL
LIN {X 0,Y 544.65,Z 479.81,A -85,B 0,C 180,E1 -3692.959,E2 -3692.959} C_VEL
LIN {X 0,Y 544.684,Z 476.895,A -85,B 0,C 180,E1 -3694.069,E2 -3694.069} C_VEL
LIN {X 0,Y 544.653,Z 472.948,A -85,B 0,C 180,E1 -3695.182,E2 -3695.182} C_VEL
LIN {X 0,Y 544.738,Z 467.712,A -85,B 0,C 180,E1 -3696.326,E2 -3696.326} C_VEL
LIN {X 0,Y 544.836,Z 461.456,A -85,B 0,C 180,E1 -3697.411,E2 -3697.411} C_VEL
LIN {X 0,Y 545.007,Z 453.43,A -85,B 0,C 180,E1 -3698.528,E2 -3698.528} C_VEL
LIN {X 0,Y 545.126,Z 445.249,A -85,B 0,C 180,E1 -3699.461,E2 -3699.461} C_VEL
LIN {X 0,Y 545.372,Z 435.275,A -85,B 0,C 180,E1 -3700.394,E2 -3700.394} C_VEL
LIN {X 0,Y 545.571,Z 424.437,A -85,B 0,C 180,E1 -3701.207,E2 -3701.207} C_VEL
LIN {X 0,Y 545.712,Z 412.976,A -85,B 0,C 180,E1 -3701.891,E2 -3701.891} C_VEL
LIN {X 0,Y 545.906,Z 400.747,A -85,B 0,C 180,E1 -3702.453,E2 -3702.453} C_VEL
LIN {X 0,Y 546.106,Z 387.923,A -85,B 0,C 180,E1 -3702.874,E2 -3702.874} C_VEL
LIN {X 0,Y 546.228,Z 374.327,A -85,B 0,C 180,E1 -3703.154,E2 -3703.154} C_VEL
LIN {X 0,Y 546.442,Z 277.789,A -85,B 0,C 180,E1 -3704.432,E2 -3704.432} C_VEL
LIN {X 0,Y 545.338,Z 270.516,A -85,B 0,C 180,E1 -3704.566,E2 -3704.566} C_VEL
LIN {X 0,Y 545.597,Z 249.483,A -85,B 0,C 180,E1 -3707.733,E2 -3707.733} C_VEL
LIN {X 0,Y 546.013,Z 229.823,A -85,B 0,C 180,E1 -3710.73,E2 -3710.73} C_VEL
LIN {X 0,Y 546.059,Z 217.042,A -85,B 0,C 180,E1 -3712.713,E2 -3712.713} C_VEL
LIN {X 0,Y 545.056,Z 211.594,A -85,B 0,C 180,E1 -3713.643,E2 -3713.643} C_VEL
LIN {X 0,Y 545.063,Z 211.589,A -85,B 0,C 180,E1 -3716.001,E2 -3716.001} C_VEL
LIN {X 0,Y 545.075,Z 211.586,A -85,B 0,C 180,E1 -3718.745,E2 -3718.745} C_VEL
LIN {X 0,Y 545.06,Z 211.592,A -85,B 0,C 180,E1 -3721.679,E2 -3721.679} C_VEL
LIN {X 0,Y 545.062,Z 211.585,A -85,B 0,C 180,E1 -3724.564,E2 -3724.564} C_VEL
LIN {X 0,Y 545.032,Z 211.595,A -85,B 0,C 180,E1 -3727.304,E2 -3727.304} C_VEL
LIN {X 0,Y 545.066,Z 211.585,A -85,B 0,C 180,E1 -3730.143,E2 -3730.143} C_VEL
LIN {X 0,Y 545.049,Z 211.587,A -85,B 0,C 180,E1 -3732.695,E2 -3732.695} C_VEL
LIN {X 0,Y 545.026,Z 211.594,A -85,B 0,C 180,E1 -3735.171,E2 -3735.171} C_VEL
LIN {X 0,Y 545.077,Z 211.583,A -85,B 0,C 180,E1 -3738.403,E2 -3738.403} C_VEL
LIN {X 0,Y 545.079,Z 211.583,A -85,B 0,C 180,E1 -3740.818,E2 -3740.818} C_VEL
LIN {X 0,Y 545.033,Z 211.595,A -85,B 0,C 180,E1 -3743.619,E2 -3743.619} C_VEL
LIN {X 0,Y 545.051,Z 211.584,A -85,B 0,C 180,E1 -3746.327,E2 -3746.327} C_VEL
LIN {X 0,Y 545.067,Z 211.586,A -85,B 0,C 180,E1 -3748.952,E2 -3748.952} C_VEL
LIN {X 0,Y 545.076,Z 211.592,A -85,B 0,C 180,E1 -3751.506,E2 -3751.506} C_VEL
LIN {X 0,Y 545.085,Z 211.58,A -85,B 0,C 180,E1 -3754.494,E2 -3754.494} C_VEL
LIN {X 0,Y 545.037,Z 211.594,A -85,B 0,C 180,E1 -3757.242,E2 -3757.242} C_VEL
LIN {X 0,Y 545.118,Z 211.577,A -85,B 0,C 180,E1 -3760.415,E2 -3760.415} C_VEL
LIN {X 0,Y 545.063,Z 211.592,A -85,B 0,C 180,E1 -3763.521,E2 -3763.521} C_VEL
LIN {X 0,Y 545.095,Z 211.584,A -85,B 0,C 180,E1 -3765.82,E2 -3765.82} C_VEL
LIN {X 0,Y 545.119,Z 211.577,A -85,B 0,C 180,E1 -3768.849,E2 -3768.849} C_VEL
LIN {X 0,Y 545.126,Z 211.578,A -85,B 0,C 180,E1 -3771.847,E2 -3771.847} C_VEL
LIN {X 0,Y 545.2,Z 211.568,A -85,B 0,C 180,E1 -3774.823,E2 -3774.823} C_VEL
LIN {X 0,Y 545.197,Z 211.57,A -85,B 0,C 180,E1 -3777.784,E2 -3777.784} C_VEL
LIN {X 0,Y 545.206,Z 211.567,A -85,B 0,C 180,E1 -3780.739,E2 -3780.739} C_VEL
LIN {X 0,Y 545.164,Z 211.573,A -85,B 0,C 180,E1 -3782.956,E2 -3782.956} C_VEL
LIN {X 0,Y 545.168,Z 211.573,A -85,B 0,C 180,E1 -3785.92,E2 -3785.92} C_VEL
LIN {X 0,Y 545.1,Z 211.579,A -85,B 0,C 180,E1 -3788.9,E2 -3788.9} C_VEL
LIN {X 0,Y 545.106,Z 211.581,A -85,B 0,C 180,E1 -3791.905,E2 -3791.905} C_VEL
LIN {X 0,Y 545.082,Z 211.584,A -85,B 0,C 180,E1 -3794.944,E2 -3794.944} C_VEL
LIN {X 0,Y 545.061,Z 211.584,A -85,B 0,C 180,E1 -3798.027,E2 -3798.027} C_VEL
LIN {X 0,Y 545.092,Z 211.58,A -85,B 0,C 180,E1 -3800.372,E2 -3800.372} C_VEL
LIN {X 0,Y 545.078,Z 211.589,A -85,B 0,C 180,E1 -3803.56,E2 -3803.56} C_VEL
LIN {X 0,Y 545.063,Z 211.584,A -85,B 0,C 180,E1 -3806.002,E2 -3806.002} C_VEL
LIN {X 0,Y 545.075,Z 211.584,A -85,B 0,C 180,E1 -3808.745,E2 -3808.745} C_VEL
LIN {X 0,Y 545.06,Z 211.59,A -85,B 0,C 180,E1 -3811.679,E2 -3811.679} C_VEL
LIN {X 0,Y 545.063,Z 211.584,A -85,B 0,C 180,E1 -3814.565,E2 -3814.565} C_VEL
LIN {X 0,Y 545.06,Z 211.587,A -85,B 0,C 180,E1 -3816.98,E2 -3816.98} C_VEL
LIN {X 0,Y 544.353,Z 211.682,A -85,B 0,C 180,E1 -3817.597,E2 -3817.597} C_VEL
LIN {X 0,Y 541.489,Z 212.038,A -85,B 0,C 180,E1 -3818.598,E2 -3818.598} C_VEL
LIN {X 0,Y 539.103,Z 212.335,A -85,B 0,C 180,E1 -3819.403,E2 -3819.403} C_VEL
LIN {X 0,Y 538.093,Z 212.454,A -85,B 0,C 180,E1 -3820.025,E2 -3820.025} C_VEL
LIN {X 0,Y 538.017,Z 212.462,A -85,B 0,C 180,E1 -3820.236,E2 -3820.236} C_VEL
LIN {X 0,Y 538,Z 212.468,A -85,B 0,C 180,E1 -3822.984,E2 -3822.984} C_VEL
LIN {X 0,Y 538.013,Z 212.464,A -85,B 0,C 180,E1 -3825.928,E2 -3825.928} C_VEL
LIN {X 0,Y 538.051,Z 212.467,A -85,B 0,C 180,E1 -3829.253,E2 -3829.253} C_VEL
LIN {X 0,Y 537.992,Z 212.468,A -85,B 0,C 180,E1 -3832.122,E2 -3832.122} C_VEL
LIN {X 0,Y 537.996,Z 212.469,A -85,B 0,C 180,E1 -3834.915,E2 -3834.915} C_VEL
LIN {X 0,Y 538.02,Z 212.468,A -85,B 0,C 180,E1 -3837.617,E2 -3837.617} C_VEL
LIN {X 0,Y 538.016,Z 212.462,A -85,B 0,C 180,E1 -3840.239,E2 -3840.239} C_VEL
LIN {X 0,Y 538.033,Z 212.463,A -85,B 0,C 180,E1 -3842.794,E2 -3842.794} C_VEL
LIN {X 0,Y 538.083,Z 212.668,A -85,B 0,C 180,E1 -3843.895,E2 -3843.895} C_VEL
LIN {X 0,Y 538.548,Z 218.169,A -85,B 0,C 180,E1 -3844.905,E2 -3844.905} C_VEL
LIN {X 0,Y 538.305,Z 233.961,A -85,B 0,C 180,E1 -3847.752,E2 -3847.752} C_VEL
LIN {X 0,Y 538.23,Z 242.544,A -85,B 0,C 180,E1 -3849.294,E2 -3849.294} C_VEL
LIN {X 0,Y 539.698,Z 252.344,A -85,B 0,C 180,E1 -3849.478,E2 -3849.478} C_VEL
LIN {X 0,Y 539.287,Z 349.332,A -85,B 0,C 180,E1 -3850.788,E2 -3850.788} C_VEL
LIN {X 0,Y 539.135,Z 362.888,A -85,B 0,C 180,E1 -3851.128,E2 -3851.128} C_VEL
LIN {X 0,Y 538.948,Z 375.814,A -85,B 0,C 180,E1 -3851.614,E2 -3851.614} C_VEL
LIN {X 0,Y 538.798,Z 387.464,A -85,B 0,C 180,E1 -3852.214,E2 -3852.214} C_VEL
LIN {X 0,Y 538.508,Z 398.295,A -85,B 0,C 180,E1 -3852.924,E2 -3852.924} C_VEL
LIN {X 0,Y 538.303,Z 408.942,A -85,B 0,C 180,E1 -3853.795,E2 -3853.795} C_VEL
LIN {X 0,Y 538.111,Z 417.597,A -85,B 0,C 180,E1 -3854.664,E2 -3854.664} C_VEL
LIN {X 0,Y 537.904,Z 425.525,A -85,B 0,C 180,E1 -3855.626,E2 -3855.626} C_VEL
LIN {X 0,Y 537.743,Z 433.218,A -85,B 0,C 180,E1 -3856.779,E2 -3856.779} C_VEL
LIN {X 0,Y 537.675,Z 439.371,A -85,B 0,C 180,E1 -3857.928,E2 -3857.928} C_VEL
LIN {X 0,Y 537.617,Z 444.219,A -85,B 0,C 180,E1 -3859.073,E2 -3859.073} C_VEL
LIN {X 0,Y 537.574,Z 447.921,A -85,B 0,C 180,E1 -3860.215,E2 -3860.215} C_VEL
LIN {X 0,Y 537.496,Z 449.826,A -85,B 0,C 180,E1 -3860.973,E2 -3860.973} C_VEL
LIN {X 0,Y 537.513,Z 451.271,A -85,B 0,C 180,E1 -3861.731,E2 -3861.731} C_VEL
LIN {X 0,Y 537.551,Z 452.915,A -85,B 0,C 180,E1 -3863.243,E2 -3863.243} C_VEL
LIN {X 0,Y 537.52,Z 453.158,A -85,B 0,C 180,E1 -3863.996,E2 -3863.996} C_VEL
LIN {X 0,Y 537.52,Z 452.978,A -85,B 0,C 180,E1 -3864.749,E2 -3864.749} C_VEL
LIN {X 0,Y 537.562,Z 451.425,A -85,B 0,C 180,E1 -3866.252,E2 -3866.252} C_VEL
LIN {X 0,Y 537.576,Z 450.069,A -85,B 0,C 180,E1 -3867.002,E2 -3867.002} C_VEL
LIN {X 0,Y 537.585,Z 447.208,A -85,B 0,C 180,E1 -3868.127,E2 -3868.127} C_VEL
LIN {X 0,Y 537.538,Z 443.342,A -85,B 0,C 180,E1 -3869.251,E2 -3869.251} C_VEL
LIN {X 0,Y 537.699,Z 438.351,A -85,B 0,C 180,E1 -3870.374,E2 -3870.374} C_VEL
LIN {X 0,Y 537.756,Z 432.106,A -85,B 0,C 180,E1 -3871.498,E2 -3871.498} C_VEL
LIN {X 0,Y 537.961,Z 424.296,A -85,B 0,C 180,E1 -3872.621,E2 -3872.621} C_VEL
LIN {X 0,Y 538.122,Z 416.365,A -85,B 0,C 180,E1 -3873.557,E2 -3873.557} C_VEL
LIN {X 0,Y 538.308,Z 406.715,A -85,B 0,C 180,E1 -3874.493,E2 -3874.493} C_VEL
LIN {X 0,Y 538.577,Z 395.966,A -85,B 0,C 180,E1 -3875.335,E2 -3875.335} C_VEL
LIN {X 0,Y 538.813,Z 383.74,A -85,B 0,C 180,E1 -3876.084,E2 -3876.084} C_VEL
LIN {X 0,Y 539.026,Z 371.782,A -85,B 0,C 180,E1 -3876.645,E2 -3876.645} C_VEL
LIN {X 0,Y 539.241,Z 359.408,A -85,B 0,C 180,E1 -3877.065,E2 -3877.065} C_VEL
LIN {X 0,Y 539.355,Z 346.57,A -85,B 0,C 180,E1 -3877.346,E2 -3877.346} C_VEL
LIN {X 0,Y 539.628,Z 250.584,A -85,B 0,C 180,E1 -3878.637,E2 -3878.637} C_VEL
LIN {X 0,Y 538.235,Z 242.531,A -85,B 0,C 180,E1 -3878.802,E2 -3878.802} C_VEL
LIN {X 0,Y 538.473,Z 226.011,A -85,B 0,C 180,E1 -3881.795,E2 -3881.795} C_VEL
LIN {X 0,Y 538.504,Z 215.124,A -85,B 0,C 180,E1 -3883.779,E2 -3883.779} C_VEL
LIN {X 0,Y 538.087,Z 212.462,A -85,B 0,C 180,E1 -3884.32,E2 -3884.32} C_VEL
LIN {X 0,Y 538.04,Z 212.461,A -85,B 0,C 180,E1 -3887.532,E2 -3887.532} C_VEL
LIN {X 0,Y 538.041,Z 212.468,A -85,B 0,C 180,E1 -3890.651,E2 -3890.651} C_VEL
LIN {X 0,Y 538.006,Z 212.463,A -85,B 0,C 180,E1 -3893.888,E2 -3893.888} C_VEL
LIN {X 0,Y 538.038,Z 212.464,A -85,B 0,C 180,E1 -3896.367,E2 -3896.367} C_VEL
LIN {X 0,Y 538.033,Z 212.465,A -85,B 0,C 180,E1 -3898.933,E2 -3898.933} C_VEL
LIN {X 0,Y 538.013,Z 212.462,A -85,B 0,C 180,E1 -3901.887,E2 -3901.887} C_VEL
LIN {X 0,Y 538.014,Z 212.471,A -85,B 0,C 180,E1 -3904.617,E2 -3904.617} C_VEL
LIN {X 0,Y 538.002,Z 212.466,A -85,B 0,C 180,E1 -3907.169,E2 -3907.169} C_VEL
LIN {X 0,Y 538.024,Z 212.461,A -85,B 0,C 180,E1 -3909.797,E2 -3909.797} C_VEL
LIN {X 0,Y 538.021,Z 212.469,A -85,B 0,C 180,E1 -3912.786,E2 -3912.786} C_VEL
LIN {X 0,Y 538.021,Z 212.462,A -85,B 0,C 180,E1 -3915.926,E2 -3915.926} C_VEL
LIN {X 0,Y 538.05,Z 212.459,A -85,B 0,C 180,E1 -3919.253,E2 -3919.253} C_VEL
LIN {X 0,Y 537.99,Z 212.467,A -85,B 0,C 180,E1 -3922.122,E2 -3922.122} C_VEL
LIN {X 0,Y 537.996,Z 212.47,A -85,B 0,C 180,E1 -3924.915,E2 -3924.915} C_VEL
LIN {X 0,Y 538.02,Z 212.461,A -85,B 0,C 180,E1 -3927.617,E2 -3927.617} C_VEL
LIN {X 0,Y 538.015,Z 212.465,A -85,B 0,C 180,E1 -3930.238,E2 -3930.238} C_VEL
LIN {X 0,Y 538.047,Z 212.465,A -85,B 0,C 180,E1 -3932.795,E2 -3932.795} C_VEL
LIN {X 0,Y 537.997,Z 212.465,A -85,B 0,C 180,E1 -3935.29,E2 -3935.29} C_VEL
LIN {X 0,Y 538.016,Z 212.463,A -85,B 0,C 180,E1 -3938.042,E2 -3938.042} C_VEL
LIN {X 0,Y 538.081,Z 212.456,A -85,B 0,C 180,E1 -3940.148,E2 -3940.148} C_VEL
LIN {X 0,Y 538.01,Z 212.463,A -85,B 0,C 180,E1 -3943.298,E2 -3943.298} C_VEL
LIN {X 0,Y 538.053,Z 212.457,A -85,B 0,C 180,E1 -3945.63,E2 -3945.63} C_VEL
LIN {X 0,Y 538.078,Z 212.463,A -85,B 0,C 180,E1 -3948.701,E2 -3948.701} C_VEL
LIN {X 0,Y 538.062,Z 212.456,A -85,B 0,C 180,E1 -3951.739,E2 -3951.739} C_VEL
LIN {X 0,Y 538.157,Z 212.452,A -85,B 0,C 180,E1 -3954.755,E2 -3954.755} C_VEL
LIN {X 0,Y 538.167,Z 212.443,A -85,B 0,C 180,E1 -3957.755,E2 -3957.755} C_VEL
LIN {X 0,Y 538.182,Z 212.448,A -85,B 0,C 180,E1 -3960.748,E2 -3960.748} C_VEL
LIN {X 0,Y 538.135,Z 212.451,A -85,B 0,C 180,E1 -3962.994,E2 -3962.994} C_VEL
LIN {X 0,Y 538.12,Z 212.45,A -85,B 0,C 180,E1 -3965.997,E2 -3965.997} C_VEL
LIN {X 0,Y 538.06,Z 212.46,A -85,B 0,C 180,E1 -3969.018,E2 -3969.018} C_VEL
LIN {X 0,Y 538.067,Z 212.458,A -85,B 0,C 180,E1 -3972.063,E2 -3972.063} C_VEL
LIN {X 0,Y 538.045,Z 212.46,A -85,B 0,C 180,E1 -3975.144,E2 -3975.144} C_VEL
LIN {X 0,Y 538.024,Z 212.465,A -85,B 0,C 180,E1 -3978.27,E2 -3978.27} C_VEL
LIN {X 0,Y 538.038,Z 212.468,A -85,B 0,C 180,E1 -3980.651,E2 -3980.651} C_VEL
LIN {X 0,Y 538.002,Z 212.464,A -85,B 0,C 180,E1 -3983.888,E2 -3983.888} C_VEL
LIN {X 0,Y 538.035,Z 212.466,A -85,B 0,C 180,E1 -3986.367,E2 -3986.367} C_VEL
LIN {X 0,Y 538.03,Z 212.464,A -85,B 0,C 180,E1 -3988.933,E2 -3988.933} C_VEL
LIN {X 0,Y 538.01,Z 212.463,A -85,B 0,C 180,E1 -3991.887,E2 -3991.887} C_VEL
LIN {X 0,Y 538.009,Z 212.472,A -85,B 0,C 180,E1 -3994.617,E2 -3994.617} C_VEL
LIN {X 0,Y 538,Z 212.465,A -85,B 0,C 180,E1 -3997.169,E2 -3997.169} C_VEL
LIN {X 0,Y 538.011,Z 212.463,A -85,B 0,C 180,E1 -3999.798,E2 -3999.798} C_VEL
LIN {X 0,Y 538.02,Z 212.462,A -85,B 0,C 180,E1 -4001.878,E2 -4001.878} C_VEL
LIN {X 0,Y 537.998,Z 212.469,A -85,B 0,C 180,E1 -4004.863,E2 -4004.863} C_VEL
LIN {X 0,Y 538.001,Z 212.465,A -85,B 0,C 180,E1 -4007.212,E2 -4007.212} C_VEL
LIN {X 0,Y 538.022,Z 212.465,A -85,B 0,C 180,E1 -4010.203,E2 -4010.203} C_VEL
LIN {X 0,Y 538.019,Z 212.463,A -85,B 0,C 180,E1 -4013.067,E2 -4013.067} C_VEL
LIN {X 0,Y 538.019,Z 212.462,A -85,B 0,C 180,E1 -4015.827,E2 -4015.827} C_VEL
LIN {X 0,Y 538.01,Z 212.472,A -85,B 0,C 180,E1 -4018.499,E2 -4018.499} C_VEL
LIN {X 0,Y 538.02,Z 212.465,A -85,B 0,C 180,E1 -4021.098,E2 -4021.098} C_VEL
LIN {X 0,Y 538.03,Z 212.462,A -85,B 0,C 180,E1 -4023.633,E2 -4023.633} C_VEL
LIN {X 0,Y 538.044,Z 212.585,A -85,B 0,C 180,E1 -4026.237,E2 -4026.237} C_VEL
LIN {X 0,Y 539.223,Z 219.76,A -85,B 0,C 180,E1 -4027.428,E2 -4027.428} C_VEL
LIN {X 0,Y 538.873,Z 237.335,A -85,B 0,C 180,E1 -4030.178,E2 -4030.178} C_VEL
LIN {X 0,Y 538.514,Z 255.152,A -85,B 0,C 180,E1 -4032.924,E2 -4032.924} C_VEL
LIN {X 0,Y 538.282,Z 270.382,A -85,B 0,C 180,E1 -4035.247,E2 -4035.247} C_VEL
LIN {X 0,Y 539.659,Z 279.558,A -85,B 0,C 180,E1 -4035.409,E2 -4035.409} C_VEL
LIN {X 0,Y 539.312,Z 378.487,A -85,B 0,C 180,E1 -4036.746,E2 -4036.746} C_VEL
LIN {X 0,Y 539.114,Z 391.78,A -85,B 0,C 180,E1 -4037.076,E2 -4037.076} C_VEL
LIN {X 0,Y 538.93,Z 403.958,A -85,B 0,C 180,E1 -4037.527,E2 -4037.527} C_VEL
LIN {X 0,Y 538.684,Z 416.527,A -85,B 0,C 180,E1 -4038.159,E2 -4038.159} C_VEL
LIN {X 0,Y 538.502,Z 427.85,A -85,B 0,C 180,E1 -4038.901,E2 -4038.901} C_VEL
LIN {X 0,Y 538.229,Z 438.297,A -85,B 0,C 180,E1 -4039.752,E2 -4039.752} C_VEL
LIN {X 0,Y 538.054,Z 446.841,A -85,B 0,C 180,E1 -4040.603,E2 -4040.603} C_VEL
LIN {X 0,Y 537.921,Z 454.724,A -85,B 0,C 180,E1 -4041.548,E2 -4041.548} C_VEL
LIN {X 0,Y 537.754,Z 462.421,A -85,B 0,C 180,E1 -4042.679,E2 -4042.679} C_VEL
LIN {X 0,Y 537.693,Z 469.518,A -85,B 0,C 180,E1 -4043.998,E2 -4043.998} C_VEL
LIN {X 0,Y 537.54,Z 474.235,A -85,B 0,C 180,E1 -4045.125,E2 -4045.125} C_VEL
LIN {X 0,Y 537.591,Z 477.843,A -85,B 0,C 180,E1 -4046.252,E2 -4046.252} C_VEL
LIN {X 0,Y 537.551,Z 479.703,A -85,B 0,C 180,E1 -4047.002,E2 -4047.002} C_VEL
LIN {X 0,Y 537.451,Z 482.09,A -85,B 0,C 180,E1 -4048.501,E2 -4048.501} C_VEL
LIN {X 0,Y 537.442,Z 482.914,A -85,B 0,C 180,E1 -4050,E2 -4050} C_VEL
LIN {X 0,Y 537.451,Z 482.091,A -85,B 0,C 180,E1 -4051.499,E2 -4051.499} C_VEL
LIN {X 0,Y 537.551,Z 479.705,A -85,B 0,C 180,E1 -4052.998,E2 -4052.998} C_VEL
LIN {X 0,Y 537.603,Z 476.773,A -85,B 0,C 180,E1 -4054.123,E2 -4054.123} C_VEL
LIN {X 0,Y 537.587,Z 472.801,A -85,B 0,C 180,E1 -4055.251,E2 -4055.251} C_VEL
LIN {X 0,Y 537.642,Z 467.914,A -85,B 0,C 180,E1 -4056.334,E2 -4056.334} C_VEL
LIN {X 0,Y 537.755,Z 461.256,A -85,B 0,C 180,E1 -4057.51,E2 -4057.51} C_VEL
LIN {X 0,Y 537.936,Z 453.228,A -85,B 0,C 180,E1 -4058.641,E2 -4058.641} C_VEL
LIN {X 0,Y 538.091,Z 445.047,A -85,B 0,C 180,E1 -4059.586,E2 -4059.586} C_VEL
LIN {X 0,Y 538.356,Z 435.072,A -85,B 0,C 180,E1 -4060.531,E2 -4060.531} C_VEL
LIN {X 0,Y 538.561,Z 425.233,A -85,B 0,C 180,E1 -4061.288,E2 -4061.288} C_VEL
LIN {X 0,Y 538.72,Z 414.184,A -85,B 0,C 180,E1 -4061.972,E2 -4061.972} C_VEL
LIN {X 0,Y 538.944,Z 401.674,A -85,B 0,C 180,E1 -4062.569,E2 -4062.569} C_VEL
LIN {X 0,Y 539.148,Z 388.629,A -85,B 0,C 180,E1 -4063.019,E2 -4063.019} C_VEL
LIN {X 0,Y 539.306,Z 375.618,A -85,B 0,C 180,E1 -4063.302,E2 -4063.302} C_VEL
LIN {X 0,Y 539.522,Z 278.301,A -85,B 0,C 180,E1 -4064.611,E2 -4064.611} C_VEL
LIN {X 0,Y 538.321,Z 270.262,A -85,B 0,C 180,E1 -4064.768,E2 -4064.768} C_VEL
LIN {X 0,Y 538.662,Z 248.55,A -85,B 0,C 180,E1 -4068.082,E2 -4068.082} C_VEL
LIN {X 0,Y 539.005,Z 228.34,A -85,B 0,C 180,E1 -4071.213,E2 -4071.213} C_VEL
LIN {X 0,Y 539.062,Z 218.115,A -85,B 0,C 180,E1 -4072.821,E2 -4072.821} C_VEL
LIN {X 0,Y 538.008,Z 212.471,A -85,B 0,C 180,E1 -4073.794,E2 -4073.794} C_VEL
LIN {X 0,Y 538.03,Z 212.464,A -85,B 0,C 180,E1 -4076.367,E2 -4076.367} C_VEL
LIN {X 0,Y 538.032,Z 212.465,A -85,B 0,C 180,E1 -4078.933,E2 -4078.933} C_VEL
LIN {X 0,Y 538.012,Z 212.467,A -85,B 0,C 180,E1 -4081.887,E2 -4081.887} C_VEL
LIN {X 0,Y 538.012,Z 212.463,A -85,B 0,C 180,E1 -4084.617,E2 -4084.617} C_VEL
LIN {X 0,Y 538.001,Z 212.469,A -85,B 0,C 180,E1 -4087.169,E2 -4087.169} C_VEL
LIN {X 0,Y 538.022,Z 212.466,A -85,B 0,C 180,E1 -4089.797,E2 -4089.797} C_VEL
LIN {X 0,Y 538.001,Z 212.465,A -85,B 0,C 180,E1 -4092.788,E2 -4092.788} C_VEL
LIN {X 0,Y 537.999,Z 212.469,A -85,B 0,C 180,E1 -4095.137,E2 -4095.137} C_VEL
LIN {X 0,Y 538.025,Z 212.462,A -85,B 0,C 180,E1 -4098.226,E2 -4098.226} C_VEL
LIN {X 0,Y 538.011,Z 212.468,A -85,B 0,C 180,E1 -4101.169,E2 -4101.169} C_VEL
LIN {X 0,Y 537.988,Z 212.467,A -85,B 0,C 180,E1 -4104.09,E2 -4104.09} C_VEL
LIN {X 0,Y 538.032,Z 212.459,A -85,B 0,C 180,E1 -4106.727,E2 -4106.727} C_VEL
LIN {X 0,Y 538.028,Z 212.467,A -85,B 0,C 180,E1 -4109.556,E2 -4109.556} C_VEL
LIN {X 0,Y 538.015,Z 212.465,A -85,B 0,C 180,E1 -4111.949,E2 -4111.949} C_VEL
LIN {X 0,Y 538.062,Z 212.454,A -85,B 0,C 180,E1 -4114.467,E2 -4114.467} C_VEL
LIN {X 0,Y 537.994,Z 212.469,A -85,B 0,C 180,E1 -4117.738,E2 -4117.738} C_VEL
LIN {X 0,Y 538.081,Z 212.455,A -85,B 0,C 180,E1 -4120.148,E2 -4120.148} C_VEL
LIN {X 0,Y 538.011,Z 212.469,A -85,B 0,C 180,E1 -4123.299,E2 -4123.299} C_VEL
LIN {X 0,Y 538.064,Z 212.462,A -85,B 0,C 180,E1 -4125.631,E2 -4125.631} C_VEL
LIN {X 0,Y 538.078,Z 212.453,A -85,B 0,C 180,E1 -4128.702,E2 -4128.702} C_VEL
LIN {X 0,Y 538.083,Z 212.457,A -85,B 0,C 180,E1 -4131.74,E2 -4131.74} C_VEL
LIN {X 0,Y 538.12,Z 212.45,A -85,B 0,C 180,E1 -4134.003,E2 -4134.003} C_VEL
LIN {X 0,Y 538.127,Z 212.451,A -85,B 0,C 180,E1 -4137.006,E2 -4137.006} C_VEL
LIN {X 0,Y 538.174,Z 212.444,A -85,B 0,C 180,E1 -4140,E2 -4140} C_VEL
LIN {X 0,Y 538.132,Z 212.449,A -85,B 0,C 180,E1 -4142.995,E2 -4142.995} C_VEL
LIN {X 0,Y 538.119,Z 212.451,A -85,B 0,C 180,E1 -4145.997,E2 -4145.997} C_VEL
LIN {X 0,Y 538.053,Z 212.458,A -85,B 0,C 180,E1 -4149.018,E2 -4149.018} C_VEL
LIN {X 0,Y 538.065,Z 212.456,A -85,B 0,C 180,E1 -4152.063,E2 -4152.063} C_VEL
LIN {X 0,Y 538.042,Z 212.463,A -85,B 0,C 180,E1 -4155.144,E2 -4155.144} C_VEL
LIN {X 0,Y 538.014,Z 212.46,A -85,B 0,C 180,E1 -4158.271,E2 -4158.271} C_VEL
LIN {X 0,Y 538.038,Z 212.459,A -85,B 0,C 180,E1 -4160.652,E2 -4160.652} C_VEL
LIN {X 0,Y 538.008,Z 212.466,A -85,B 0,C 180,E1 -4163.878,E2 -4163.878} C_VEL
LIN {X 0,Y 538.03,Z 212.458,A -85,B 0,C 180,E1 -4166.368,E2 -4166.368} C_VEL
LIN {X 0,Y 538.032,Z 212.463,A -85,B 0,C 180,E1 -4168.933,E2 -4168.933} C_VEL
LIN {X 0,Y 538.012,Z 212.465,A -85,B 0,C 180,E1 -4171.887,E2 -4171.887} C_VEL
LIN {X 0,Y 538.012,Z 212.463,A -85,B 0,C 180,E1 -4174.617,E2 -4174.617} C_VEL
LIN {X 0,Y 538.001,Z 212.469,A -85,B 0,C 180,E1 -4177.169,E2 -4177.169} C_VEL
LIN {X 0,Y 538.017,Z 212.462,A -85,B 0,C 180,E1 -4180.236,E2 -4180.236} C_VEL
LIN {X 0,Y 537.366,Z 212.546,A -85,B 0,C 180,E1 -4180.861,E2 -4180.861} C_VEL
LIN {X 0,Y 534.509,Z 212.909,A -85,B 0,C 180,E1 -4181.876,E2 -4181.876} C_VEL
LIN {X 0,Y 532.081,Z 213.216,A -85,B 0,C 180,E1 -4182.693,E2 -4182.693} C_VEL
LIN {X 0,Y 531.033,Z 213.343,A -85,B 0,C 180,E1 -4183.324,E2 -4183.324} C_VEL
LIN {X 0,Y 530.945,Z 213.351,A -85,B 0,C 180,E1 -4183.538,E2 -4183.538} C_VEL
LIN {X 0,Y 530.939,Z 213.343,A -85,B 0,C 180,E1 -4186.503,E2 -4186.503} C_VEL
LIN {X 0,Y 530.984,Z 213.343,A -85,B 0,C 180,E1 -4188.977,E2 -4188.977} C_VEL
LIN {X 0,Y 530.958,Z 213.351,A -85,B 0,C 180,E1 -4191.529,E2 -4191.529} C_VEL
LIN {X 0,Y 530.952,Z 213.344,A -85,B 0,C 180,E1 -4194.38,E2 -4194.38} C_VEL
LIN {X 0,Y 530.969,Z 213.347,A -85,B 0,C 180,E1 -4197.134,E2 -4197.134} C_VEL
LIN {X 0,Y 530.971,Z 213.342,A -85,B 0,C 180,E1 -4199.803,E2 -4199.803} C_VEL
LIN {X 0,Y 530.976,Z 213.341,A -85,B 0,C 180,E1 -4202.476,E2 -4202.476} C_VEL
LIN {X 0,Y 531.046,Z 213.466,A -85,B 0,C 180,E1 -4203.77,E2 -4203.77} C_VEL
LIN {X 0,Y 531.555,Z 218.796,A -85,B 0,C 180,E1 -4204.761,E2 -4204.761} C_VEL
LIN {X 0,Y 531.314,Z 234.884,A -85,B 0,C 180,E1 -4207.682,E2 -4207.682} C_VEL
LIN {X 0,Y 531.195,Z 242.71,A -85,B 0,C 180,E1 -4209.099,E2 -4209.099} C_VEL
LIN {X 0,Y 532.837,Z 252.874,A -85,B 0,C 180,E1 -4209.291,E2 -4209.291} C_VEL
LIN {X 0,Y 532.38,Z 350.281,A -85,B 0,C 180,E1 -4210.629,E2 -4210.629} C_VEL
LIN {X 0,Y 532.232,Z 363.59,A -85,B 0,C 180,E1 -4210.974,E2 -4210.974} C_VEL
LIN {X 0,Y 532.012,Z 376.362,A -85,B 0,C 180,E1 -4211.466,E2 -4211.466} C_VEL
LIN {X 0,Y 531.794,Z 388.999,A -85,B 0,C 180,E1 -4212.138,E2 -4212.138} C_VEL
LIN {X 0,Y 531.506,Z 400.018,A -85,B 0,C 180,E1 -4212.89,E2 -4212.89} C_VEL
LIN {X 0,Y 531.265,Z 410.36,A -85,B 0,C 180,E1 -4213.772,E2 -4213.772} C_VEL
LIN {X 0,Y 531.049,Z 420.065,A -85,B 0,C 180,E1 -4214.804,E2 -4214.804} C_VEL
LIN {X 0,Y 530.846,Z 427.899,A -85,B 0,C 180,E1 -4215.823,E2 -4215.823} C_VEL
LIN {X 0,Y 530.683,Z 435.2,A -85,B 0,C 180,E1 -4216.989,E2 -4216.989} C_VEL
LIN {X 0,Y 530.592,Z 440.988,A -85,B 0,C 180,E1 -4218.153,E2 -4218.153} C_VEL
LIN {X 0,Y 530.497,Z 445.515,A -85,B 0,C 180,E1 -4219.311,E2 -4219.311} C_VEL
LIN {X 0,Y 530.478,Z 447.893,A -85,B 0,C 180,E1 -4220.083,E2 -4220.083} C_VEL
LIN {X 0,Y 530.409,Z 449.835,A -85,B 0,C 180,E1 -4220.851,E2 -4220.851} C_VEL
LIN {X 0,Y 530.427,Z 451.347,A -85,B 0,C 180,E1 -4221.619,E2 -4221.619} C_VEL
LIN {X 0,Y 530.467,Z 453.061,A -85,B 0,C 180,E1 -4223.152,E2 -4223.152} C_VEL
LIN {X 0,Y 530.443,Z 453.221,A -85,B 0,C 180,E1 -4224.678,E2 -4224.678} C_VEL
LIN {X 0,Y 530.48,Z 451.738,A -85,B 0,C 180,E1 -4226.202,E2 -4226.202} C_VEL
LIN {X 0,Y 530.478,Z 450.417,A -85,B 0,C 180,E1 -4226.962,E2 -4226.962} C_VEL
LIN {X 0,Y 530.511,Z 447.624,A -85,B 0,C 180,E1 -4228.102,E2 -4228.102} C_VEL
LIN {X 0,Y 530.453,Z 443.833,A -85,B 0,C 180,E1 -4229.241,E2 -4229.241} C_VEL
LIN {X 0,Y 530.63,Z 438.921,A -85,B 0,C 180,E1 -4230.379,E2 -4230.379} C_VEL
LIN {X 0,Y 530.691,Z 432.774,A -85,B 0,C 180,E1 -4231.518,E2 -4231.518} C_VEL
LIN {X 0,Y 530.911,Z 425.106,A -85,B 0,C 180,E1 -4232.656,E2 -4232.656} C_VEL
LIN {X 0,Y 531.092,Z 417.295,A -85,B 0,C 180,E1 -4233.604,E2 -4233.604} C_VEL
LIN {X 0,Y 531.334,Z 406.736,A -85,B 0,C 180,E1 -4234.647,E2 -4234.647} C_VEL
LIN {X 0,Y 531.629,Z 395.932,A -85,B 0,C 180,E1 -4235.5,E2 -4235.5} C_VEL
LIN {X 0,Y 531.893,Z 383.645,A -85,B 0,C 180,E1 -4236.258,E2 -4236.258} C_VEL
LIN {X 0,Y 532.117,Z 371.607,A -85,B 0,C 180,E1 -4236.827,E2 -4236.827} C_VEL
LIN {X 0,Y 532.34,Z 359.007,A -85,B 0,C 180,E1 -4237.253,E2 -4237.253} C_VEL
LIN {X 0,Y 532.47,Z 345.78,A -85,B 0,C 180,E1 -4237.537,E2 -4237.537} C_VEL
LIN {X 0,Y 532.776,Z 251.382,A -85,B 0,C 180,E1 -4238.821,E2 -4238.821} C_VEL
LIN {X 0,Y 531.229,Z 242.732,A -85,B 0,C 180,E1 -4238.991,E2 -4238.991} C_VEL
LIN {X 0,Y 531.483,Z 226.824,A -85,B 0,C 180,E1 -4241.893,E2 -4241.893} C_VEL
LIN {X 0,Y 531.568,Z 216.632,A -85,B 0,C 180,E1 -4243.767,E2 -4243.767} C_VEL
LIN {X 0,Y 531.051,Z 213.339,A -85,B 0,C 180,E1 -4244.416,E2 -4244.416} C_VEL
LIN {X 0,Y 530.985,Z 213.34,A -85,B 0,C 180,E1 -4247.723,E2 -4247.723} C_VEL
LIN {X 0,Y 531.029,Z 213.334,A -85,B 0,C 180,E1 -4250.127,E2 -4250.127} C_VEL
LIN {X 0,Y 530.949,Z 213.35,A -85,B 0,C 180,E1 -4252.573,E2 -4252.573} C_VEL
LIN {X 0,Y 531.002,Z 213.339,A -85,B 0,C 180,E1 -4255.058,E2 -4255.058} C_VEL
LIN {X 0,Y 530.973,Z 213.339,A -85,B 0,C 180,E1 -4257.598,E2 -4257.598} C_VEL
LIN {X 0,Y 530.971,Z 213.342,A -85,B 0,C 180,E1 -4260.197,E2 -4260.197} C_VEL
LIN {X 0,Y 530.969,Z 213.346,A -85,B 0,C 180,E1 -4262.866,E2 -4262.866} C_VEL
LIN {X 0,Y 530.953,Z 213.342,A -85,B 0,C 180,E1 -4265.62,E2 -4265.62} C_VEL
LIN {X 0,Y 530.967,Z 213.349,A -85,B 0,C 180,E1 -4268.653,E2 -4268.653} C_VEL
LIN {X 0,Y 530.995,Z 213.337,A -85,B 0,C 180,E1 -4271.435,E2 -4271.435} C_VEL
LIN {X 0,Y 530.976,Z 213.346,A -85,B 0,C 180,E1 -4274.548,E2 -4274.548} C_VEL
LIN {X 0,Y 530.974,Z 213.339,A -85,B 0,C 180,E1 -4277.835,E2 -4277.835} C_VEL
LIN {X 0,Y 530.986,Z 213.345,A -85,B 0,C 180,E1 -4280.556,E2 -4280.556} C_VEL
LIN {X 0,Y 530.952,Z 213.342,A -85,B 0,C 180,E1 -4283.441,E2 -4283.441} C_VEL
LIN {X 0,Y 531,Z 213.343,A -85,B 0,C 180,E1 -4286.494,E2 -4286.494} C_VEL
LIN {X 0,Y 530.975,Z 213.34,A -85,B 0,C 180,E1 -4289.355,E2 -4289.355} C_VEL
LIN {X 0,Y 531.009,Z 213.341,A -85,B 0,C 180,E1 -4292.468,E2 -4292.468} C_VEL
LIN {X 0,Y 530.963,Z 213.345,A -85,B 0,C 180,E1 -4294.94,E2 -4294.94} C_VEL
LIN {X 0,Y 530.978,Z 213.339,A -85,B 0,C 180,E1 -4297.898,E2 -4297.898} C_VEL
LIN {X 0,Y 530.986,Z 213.347,A -85,B 0,C 180,E1 -4300.677,E2 -4300.677} C_VEL
LIN {X 0,Y 530.969,Z 213.343,A -85,B 0,C 180,E1 -4303.07,E2 -4303.07} C_VEL
LIN {X 0,Y 531.01,Z 213.335,A -85,B 0,C 180,E1 -4305.435,E2 -4305.435} C_VEL
LIN {X 0,Y 531.036,Z 213.34,A -85,B 0,C 180,E1 -4308.55,E2 -4308.55} C_VEL
LIN {X 0,Y 531.036,Z 213.331,A -85,B 0,C 180,E1 -4311.629,E2 -4311.629} C_VEL
LIN {X 0,Y 531.117,Z 213.33,A -85,B 0,C 180,E1 -4314.685,E2 -4314.685} C_VEL
LIN {X 0,Y 531.139,Z 213.318,A -85,B 0,C 180,E1 -4317.725,E2 -4317.725} C_VEL
LIN {X 0,Y 531.152,Z 213.324,A -85,B 0,C 180,E1 -4320.758,E2 -4320.758} C_VEL
LIN {X 0,Y 531.101,Z 213.326,A -85,B 0,C 180,E1 -4323.034,E2 -4323.034} C_VEL
LIN {X 0,Y 531.081,Z 213.328,A -85,B 0,C 180,E1 -4326.077,E2 -4326.077} C_VEL
LIN {X 0,Y 531.052,Z 213.335,A -85,B 0,C 180,E1 -4328.371,E2 -4328.371} C_VEL
LIN {X 0,Y 531.051,Z 213.329,A -85,B 0,C 180,E1 -4331.671,E2 -4331.671} C_VEL
LIN {X 0,Y 531.032,Z 213.336,A -85,B 0,C 180,E1 -4334.956,E2 -4334.956} C_VEL
LIN {X 0,Y 530.982,Z 213.338,A -85,B 0,C 180,E1 -4337.724,E2 -4337.724} C_VEL
LIN {X 0,Y 531.025,Z 213.335,A -85,B 0,C 180,E1 -4340.127,E2 -4340.127} C_VEL
LIN {X 0,Y 530.945,Z 213.352,A -85,B 0,C 180,E1 -4342.573,E2 -4342.573} C_VEL
LIN {X 0,Y 530.999,Z 213.338,A -85,B 0,C 180,E1 -4345.058,E2 -4345.058} C_VEL
LIN {X 0,Y 530.97,Z 213.339,A -85,B 0,C 180,E1 -4347.598,E2 -4347.598} C_VEL
LIN {X 0,Y 530.969,Z 213.344,A -85,B 0,C 180,E1 -4350.197,E2 -4350.197} C_VEL
LIN {X 0,Y 530.967,Z 213.345,A -85,B 0,C 180,E1 -4352.867,E2 -4352.867} C_VEL
LIN {X 0,Y 530.95,Z 213.342,A -85,B 0,C 180,E1 -4355.62,E2 -4355.62} C_VEL
LIN {X 0,Y 530.965,Z 213.348,A -85,B 0,C 180,E1 -4358.653,E2 -4358.653} C_VEL
LIN {X 0,Y 530.99,Z 213.337,A -85,B 0,C 180,E1 -4361.436,E2 -4361.436} C_VEL
LIN {X 0,Y 530.968,Z 213.35,A -85,B 0,C 180,E1 -4364.549,E2 -4364.549} C_VEL
LIN {X 0,Y 530.973,Z 213.34,A -85,B 0,C 180,E1 -4367.836,E2 -4367.836} C_VEL
LIN {X 0,Y 530.985,Z 213.347,A -85,B 0,C 180,E1 -4370.557,E2 -4370.557} C_VEL
LIN {X 0,Y 530.951,Z 213.342,A -85,B 0,C 180,E1 -4373.441,E2 -4373.441} C_VEL
LIN {X 0,Y 531,Z 213.345,A -85,B 0,C 180,E1 -4376.494,E2 -4376.494} C_VEL
LIN {X 0,Y 530.967,Z 213.34,A -85,B 0,C 180,E1 -4379.357,E2 -4379.357} C_VEL
LIN {X 0,Y 531.009,Z 213.344,A -85,B 0,C 180,E1 -4382.469,E2 -4382.469} C_VEL
LIN {X 0,Y 530.962,Z 213.345,A -85,B 0,C 180,E1 -4384.94,E2 -4384.94} C_VEL
LIN {X 0,Y 530.976,Z 213.457,A -85,B 0,C 180,E1 -4386.076,E2 -4386.076} C_VEL
LIN {X 0,Y 532.239,Z 220.588,A -85,B 0,C 180,E1 -4387.28,E2 -4387.28} C_VEL
LIN {X 0,Y 531.92,Z 237.147,A -85,B 0,C 180,E1 -4389.908,E2 -4389.908} C_VEL
LIN {X 0,Y 531.551,Z 253.686,A -85,B 0,C 180,E1 -4392.495,E2 -4392.495} C_VEL
LIN {X 0,Y 531.265,Z 270.151,A -85,B 0,C 180,E1 -4395.043,E2 -4395.043} C_VEL
LIN {X 0,Y 532.787,Z 280.633,A -85,B 0,C 180,E1 -4395.234,E2 -4395.234} C_VEL
LIN {X 0,Y 532.424,Z 378.282,A -85,B 0,C 180,E1 -4396.571,E2 -4396.571} C_VEL
LIN {X 0,Y 532.207,Z 390.815,A -85,B 0,C 180,E1 -4396.881,E2 -4396.881} C_VEL
LIN {X 0,Y 531.966,Z 403.756,A -85,B 0,C 180,E1 -4397.361,E2 -4397.361} C_VEL
LIN {X 0,Y 531.695,Z 416.281,A -85,B 0,C 180,E1 -4397.999,E2 -4397.999} C_VEL
LIN {X 0,Y 531.507,Z 427.651,A -85,B 0,C 180,E1 -4398.753,E2 -4398.753} C_VEL
LIN {X 0,Y 531.213,Z 438.099,A -85,B 0,C 180,E1 -4399.615,E2 -4399.615} C_VEL
LIN {X 0,Y 531.028,Z 446.643,A -85,B 0,C 180,E1 -4400.478,E2 -4400.478} C_VEL
LIN {X 0,Y 530.869,Z 454.526,A -85,B 0,C 180,E1 -4401.435,E2 -4401.435} C_VEL
LIN {X 0,Y 530.668,Z 462.223,A -85,B 0,C 180,E1 -4402.581,E2 -4402.581} C_VEL
LIN {X 0,Y 530.583,Z 469.32,A -85,B 0,C 180,E1 -4403.917,E2 -4403.917} C_VEL
LIN {X 0,Y 530.459,Z 474.039,A -85,B 0,C 180,E1 -4405.06,E2 -4405.06} C_VEL
LIN {X 0,Y 530.516,Z 477.648,A -85,B 0,C 180,E1 -4406.202,E2 -4406.202} C_VEL
LIN {X 0,Y 530.457,Z 479.506,A -85,B 0,C 180,E1 -4406.962,E2 -4406.962} C_VEL
LIN {X 0,Y 530.411,Z 480.9,A -85,B 0,C 180,E1 -4407.722,E2 -4407.722} C_VEL
LIN {X 0,Y 530.345,Z 482.501,A -85,B 0,C 180,E1 -4409.241,E2 -4409.241} C_VEL
LIN {X 0,Y 530.346,Z 482.717,A -85,B 0,C 180,E1 -4410,E2 -4410} C_VEL
LIN {X 0,Y 530.361,Z 481.895,A -85,B 0,C 180,E1 -4411.519,E2 -4411.519} C_VEL
LIN {X 0,Y 530.411,Z 480.902,A -85,B 0,C 180,E1 -4412.278,E2 -4412.278} C_VEL
LIN {X 0,Y 530.457,Z 479.508,A -85,B 0,C 180,E1 -4413.038,E2 -4413.038} C_VEL
LIN {X 0,Y 530.522,Z 476.576,A -85,B 0,C 180,E1 -4414.178,E2 -4414.178} C_VEL
LIN {X 0,Y 530.524,Z 472.603,A -85,B 0,C 180,E1 -4415.321,E2 -4415.321} C_VEL
LIN {X 0,Y 530.56,Z 467.079,A -85,B 0,C 180,E1 -4416.546,E2 -4416.546} C_VEL
LIN {X 0,Y 530.688,Z 461.055,A -85,B 0,C 180,E1 -4417.61,E2 -4417.61} C_VEL
LIN {X 0,Y 530.865,Z 453.027,A -85,B 0,C 180,E1 -4418.757,E2 -4418.757} C_VEL
LIN {X 0,Y 531.061,Z 444.846,A -85,B 0,C 180,E1 -4419.714,E2 -4419.714} C_VEL
LIN {X 0,Y 531.331,Z 434.87,A -85,B 0,C 180,E1 -4420.672,E2 -4420.672} C_VEL
LIN {X 0,Y 531.576,Z 425.03,A -85,B 0,C 180,E1 -4421.439,E2 -4421.439} C_VEL
LIN {X 0,Y 531.746,Z 414.552,A -85,B 0,C 180,E1 -4422.1,E2 -4422.1} C_VEL
LIN {X 0,Y 532.001,Z 401.469,A -85,B 0,C 180,E1 -4422.735,E2 -4422.735} C_VEL
LIN {X 0,Y 532.238,Z 388.421,A -85,B 0,C 180,E1 -4423.191,E2 -4423.191} C_VEL
LIN {X 0,Y 532.414,Z 375.405,A -85,B 0,C 180,E1 -4423.478,E2 -4423.478} C_VEL
LIN {X 0,Y 532.683,Z 279.164,A -85,B 0,C 180,E1 -4424.789,E2 -4424.789} C_VEL
LIN {X 0,Y 531.281,Z 270.027,A -85,B 0,C 180,E1 -4424.973,E2 -4424.973} C_VEL
LIN {X 0,Y 531.643,Z 249.772,A -85,B 0,C 180,E1 -4428.106,E2 -4428.106} C_VEL
LIN {X 0,Y 532.022,Z 230.69,A -85,B 0,C 180,E1 -4431.098,E2 -4431.098} C_VEL
LIN {X 0,Y 532.253,Z 220.471,A -85,B 0,C 180,E1 -4432.72,E2 -4432.72} C_VEL
LIN {X 0,Y 530.959,Z 213.349,A -85,B 0,C 180,E1 -4433.948,E2 -4433.948} C_VEL
LIN {X 0,Y 530.987,Z 213.342,A -85,B 0,C 180,E1 -4436.745,E2 -4436.745} C_VEL
LIN {X 0,Y 530.982,Z 213.346,A -85,B 0,C 180,E1 -4439.323,E2 -4439.323} C_VEL
LIN {X 0,Y 530.967,Z 213.343,A -85,B 0,C 180,E1 -4442.1,E2 -4442.1} C_VEL
LIN {X 0,Y 530.969,Z 213.342,A -85,B 0,C 180,E1 -4444.851,E2 -4444.851} C_VEL
LIN {X 0,Y 530.964,Z 213.35,A -85,B 0,C 180,E1 -4447.508,E2 -4447.508} C_VEL
LIN {X 0,Y 530.982,Z 213.339,A -85,B 0,C 180,E1 -4450.433,E2 -4450.433} C_VEL
LIN {X 0,Y 530.946,Z 213.352,A -85,B 0,C 180,E1 -4453.497,E2 -4453.497} C_VEL
LIN {X 0,Y 530.938,Z 213.344,A -85,B 0,C 180,E1 -4456.502,E2 -4456.502} C_VEL
LIN {X 0,Y 530.983,Z 213.341,A -85,B 0,C 180,E1 -4458.977,E2 -4458.977} C_VEL
LIN {X 0,Y 530.954,Z 213.35,A -85,B 0,C 180,E1 -4461.529,E2 -4461.529} C_VEL
LIN {X 0,Y 530.949,Z 213.342,A -85,B 0,C 180,E1 -4464.379,E2 -4464.379} C_VEL
LIN {X 0,Y 530.967,Z 213.343,A -85,B 0,C 180,E1 -4467.133,E2 -4467.133} C_VEL
LIN {X 0,Y 530.969,Z 213.342,A -85,B 0,C 180,E1 -4469.803,E2 -4469.803} C_VEL
LIN {X 0,Y 530.973,Z 213.339,A -85,B 0,C 180,E1 -4472.476,E2 -4472.476} C_VEL
LIN {X 0,Y 530.989,Z 213.338,A -85,B 0,C 180,E1 -4474.942,E2 -4474.942} C_VEL
LIN {X 0,Y 530.972,Z 213.338,A -85,B 0,C 180,E1 -4478.247,E2 -4478.247} C_VEL
LIN {X 0,Y 530.992,Z 213.337,A -85,B 0,C 180,E1 -4480.677,E2 -4480.677} C_VEL
LIN {X 0,Y 530.97,Z 213.343,A -85,B 0,C 180,E1 -4483.07,E2 -4483.07} C_VEL
LIN {X 0,Y 531.042,Z 213.34,A -85,B 0,C 180,E1 -4485.437,E2 -4485.437} C_VEL
LIN {X 0,Y 531.036,Z 213.329,A -85,B 0,C 180,E1 -4488.55,E2 -4488.55} C_VEL
LIN {X 0,Y 531.052,Z 213.334,A -85,B 0,C 180,E1 -4491.629,E2 -4491.629} C_VEL
LIN {X 0,Y 531.117,Z 213.321,A -85,B 0,C 180,E1 -4494.685,E2 -4494.685} C_VEL
LIN {X 0,Y 531.14,Z 213.321,A -85,B 0,C 180,E1 -4497.725,E2 -4497.725} C_VEL
LIN {X 0,Y 531.148,Z 213.318,A -85,B 0,C 180,E1 -4500.758,E2 -4500.758} C_VEL
LIN {X 0,Y 531.099,Z 213.326,A -85,B 0,C 180,E1 -4503.034,E2 -4503.034} C_VEL
LIN {X 0,Y 531.073,Z 213.328,A -85,B 0,C 180,E1 -4506.077,E2 -4506.077} C_VEL
LIN {X 0,Y 531.015,Z 213.336,A -85,B 0,C 180,E1 -4509.139,E2 -4509.139} C_VEL
LIN {X 0,Y 531.051,Z 213.334,A -85,B 0,C 180,E1 -4511.671,E2 -4511.671} C_VEL
LIN {X 0,Y 531.024,Z 213.335,A -85,B 0,C 180,E1 -4514.952,E2 -4514.952} C_VEL
LIN {X 0,Y 530.981,Z 213.341,A -85,B 0,C 180,E1 -4517.724,E2 -4517.724} C_VEL
LIN {X 0,Y 531.026,Z 213.333,A -85,B 0,C 180,E1 -4520.127,E2 -4520.127} C_VEL
LIN {X 0,Y 530.945,Z 213.34,A -85,B 0,C 180,E1 -4522.574,E2 -4522.574} C_VEL
LIN {X 0,Y 530.963,Z 213.345,A -85,B 0,C 180,E1 -4525.06,E2 -4525.06} C_VEL
LIN {X 0,Y 531.009,Z 213.342,A -85,B 0,C 180,E1 -4527.596,E2 -4527.596} C_VEL
LIN {X 0,Y 530.968,Z 213.339,A -85,B 0,C 180,E1 -4530.644,E2 -4530.644} C_VEL
LIN {X 0,Y 530.988,Z 213.342,A -85,B 0,C 180,E1 -4533.773,E2 -4533.773} C_VEL
LIN {X 0,Y 530.952,Z 213.341,A -85,B 0,C 180,E1 -4536.559,E2 -4536.559} C_VEL
LIN {X 0,Y 530.986,Z 213.346,A -85,B 0,C 180,E1 -4539.444,E2 -4539.444} C_VEL
LIN {X 0,Y 530.967,Z 213.341,A -85,B 0,C 180,E1 -4542.458,E2 -4542.458} C_VEL
LIN {X 0,Y 530.945,Z 213.351,A -85,B 0,C 180,E1 -4543.538,E2 -4543.538} C_VEL
LIN {X 0,Y 530.272,Z 213.43,A -85,B 0,C 180,E1 -4544.171,E2 -4544.171} C_VEL
LIN {X 0,Y 527.417,Z 213.79,A -85,B 0,C 180,E1 -4545.2,E2 -4545.2} C_VEL
LIN {X 0,Y 525.009,Z 214.085,A -85,B 0,C 180,E1 -4546.028,E2 -4546.028} C_VEL
LIN {X 0,Y 523.976,Z 214.211,A -85,B 0,C 180,E1 -4546.668,E2 -4546.668} C_VEL
LIN {X 0,Y 523.893,Z 214.222,A -85,B 0,C 180,E1 -4546.884,E2 -4546.884} C_VEL
LIN {X 0,Y 523.939,Z 214.22,A -85,B 0,C 180,E1 -4548.908,E2 -4548.908} C_VEL
LIN {X 0,Y 523.916,Z 214.223,A -85,B 0,C 180,E1 -4551.898,E2 -4551.898} C_VEL
LIN {X 0,Y 523.925,Z 214.222,A -85,B 0,C 180,E1 -4554.912,E2 -4554.912} C_VEL
LIN {X 0,Y 523.938,Z 214.221,A -85,B 0,C 180,E1 -4557.68,E2 -4557.68} C_VEL
LIN {X 0,Y 523.956,Z 214.214,A -85,B 0,C 180,E1 -4560.677,E2 -4560.677} C_VEL
LIN {X 0,Y 523.97,Z 214.326,A -85,B 0,C 180,E1 -4563.648,E2 -4563.648} C_VEL
LIN {X 0,Y 524.589,Z 219.423,A -85,B 0,C 180,E1 -4564.614,E2 -4564.614} C_VEL
LIN {X 0,Y 524.311,Z 236.042,A -85,B 0,C 180,E1 -4567.653,E2 -4567.653} C_VEL
LIN {X 0,Y 524.204,Z 242.858,A -85,B 0,C 180,E1 -4568.891,E2 -4568.891} C_VEL
LIN {X 0,Y 525.998,Z 253.65,A -85,B 0,C 180,E1 -4569.102,E2 -4569.102} C_VEL
LIN {X 0,Y 525.491,Z 350.061,A -85,B 0,C 180,E1 -4570.441,E2 -4570.441} C_VEL
LIN {X 0,Y 525.327,Z 363.506,A -85,B 0,C 180,E1 -4570.79,E2 -4570.79} C_VEL
LIN {X 0,Y 525.125,Z 375.8,A -85,B 0,C 180,E1 -4571.264,E2 -4571.264} C_VEL
LIN {X 0,Y 524.961,Z 386.479,A -85,B 0,C 180,E1 -4571.814,E2 -4571.814} C_VEL
LIN {X 0,Y 524.597,Z 397.793,A -85,B 0,C 180,E1 -4572.557,E2 -4572.557} C_VEL
LIN {X 0,Y 524.367,Z 408.598,A -85,B 0,C 180,E1 -4573.452,E2 -4573.452} C_VEL
LIN {X 0,Y 524.085,Z 418.276,A -85,B 0,C 180,E1 -4574.443,E2 -4574.443} C_VEL
LIN {X 0,Y 523.827,Z 426.144,A -85,B 0,C 180,E1 -4575.43,E2 -4575.43} C_VEL
LIN {X 0,Y 523.643,Z 433.794,A -85,B 0,C 180,E1 -4576.613,E2 -4576.613} C_VEL
LIN {X 0,Y 523.538,Z 440.825,A -85,B 0,C 180,E1 -4577.991,E2 -4577.991} C_VEL
LIN {X 0,Y 523.436,Z 445.441,A -85,B 0,C 180,E1 -4579.165,E2 -4579.165} C_VEL
LIN {X 0,Y 523.399,Z 447.866,A -85,B 0,C 180,E1 -4579.947,E2 -4579.947} C_VEL
LIN {X 0,Y 523.321,Z 449.844,A -85,B 0,C 180,E1 -4580.726,E2 -4580.726} C_VEL
LIN {X 0,Y 523.336,Z 451.401,A -85,B 0,C 180,E1 -4581.505,E2 -4581.505} C_VEL
LIN {X 0,Y 523.331,Z 452.514,A -85,B 0,C 180,E1 -4582.282,E2 -4582.282} C_VEL
LIN {X 0,Y 523.36,Z 453.465,A -85,B 0,C 180,E1 -4583.577,E2 -4583.577} C_VEL
LIN {X 0,Y 523.368,Z 453.444,A -85,B 0,C 180,E1 -4584.606,E2 -4584.606} C_VEL
LIN {X 0,Y 523.305,Z 452.955,A -85,B 0,C 180,E1 -4585.378,E2 -4585.378} C_VEL
LIN {X 0,Y 523.4,Z 452.051,A -85,B 0,C 180,E1 -4586.15,E2 -4586.15} C_VEL
LIN {X 0,Y 523.384,Z 450.764,A -85,B 0,C 180,E1 -4586.921,E2 -4586.921} C_VEL
LIN {X 0,Y 523.408,Z 448.041,A -85,B 0,C 180,E1 -4588.076,E2 -4588.076} C_VEL
LIN {X 0,Y 523.368,Z 444.324,A -85,B 0,C 180,E1 -4589.231,E2 -4589.231} C_VEL
LIN {X 0,Y 523.54,Z 439.493,A -85,B 0,C 180,E1 -4590.385,E2 -4590.385} C_VEL
LIN {X 0,Y 523.624,Z 433.432,A -85,B 0,C 180,E1 -4591.538,E2 -4591.538} C_VEL
LIN {X 0,Y 523.864,Z 425.904,A -85,B 0,C 180,E1 -4592.691,E2 -4592.691} C_VEL
LIN {X 0,Y 524.064,Z 418.222,A -85,B 0,C 180,E1 -4593.652,E2 -4593.652} C_VEL
LIN {X 0,Y 524.329,Z 407.812,A -85,B 0,C 180,E1 -4594.709,E2 -4594.709} C_VEL
LIN {X 0,Y 524.649,Z 397.229,A -85,B 0,C 180,E1 -4595.573,E2 -4595.573} C_VEL
LIN {X 0,Y 524.906,Z 386.996,A -85,B 0,C 180,E1 -4596.245,E2 -4596.245} C_VEL
LIN {X 0,Y 525.134,Z 374.775,A -85,B 0,C 180,E1 -4596.87,E2 -4596.87} C_VEL
LIN {X 0,Y 525.374,Z 361.918,A -85,B 0,C 180,E1 -4597.349,E2 -4597.349} C_VEL
LIN {X 0,Y 525.538,Z 349.392,A -85,B 0,C 180,E1 -4597.661,E2 -4597.661} C_VEL
LIN {X 0,Y 525.876,Z 251.878,A -85,B 0,C 180,E1 -4599.015,E2 -4599.015} C_VEL
LIN {X 0,Y 524.24,Z 242.838,A -85,B 0,C 180,E1 -4599.204,E2 -4599.204} C_VEL
LIN {X 0,Y 524.498,Z 227.651,A -85,B 0,C 180,E1 -4601.994,E2 -4601.994} C_VEL
LIN {X 0,Y 524.632,Z 218.165,A -85,B 0,C 180,E1 -4603.756,E2 -4603.756} C_VEL
LIN {X 0,Y 524.029,Z 214.215,A -85,B 0,C 180,E1 -4604.564,E2 -4604.564} C_VEL
LIN {X 0,Y 523.951,Z 214.217,A -85,B 0,C 180,E1 -4607.969,E2 -4607.969} C_VEL
LIN {X 0,Y 523.976,Z 214.216,A -85,B 0,C 180,E1 -4610.41,E2 -4610.41} C_VEL
LIN {X 0,Y 523.914,Z 214.225,A -85,B 0,C 180,E1 -4612.893,E2 -4612.893} C_VEL
LIN {X 0,Y 523.938,Z 214.216,A -85,B 0,C 180,E1 -4615.419,E2 -4615.419} C_VEL
LIN {X 0,Y 523.92,Z 214.219,A -85,B 0,C 180,E1 -4618.002,E2 -4618.002} C_VEL
LIN {X 0,Y 523.948,Z 214.221,A -85,B 0,C 180,E1 -4620.854,E2 -4620.854} C_VEL
LIN {X 0,Y 523.962,Z 214.213,A -85,B 0,C 180,E1 -4623.734,E2 -4623.734} C_VEL
LIN {X 0,Y 523.901,Z 214.225,A -85,B 0,C 180,E1 -4626.4,E2 -4626.4} C_VEL
LIN {X 0,Y 523.921,Z 214.221,A -85,B 0,C 180,E1 -4629.085,E2 -4629.085} C_VEL
LIN {X 0,Y 523.953,Z 214.216,A -85,B 0,C 180,E1 -4632.119,E2 -4632.119} C_VEL
LIN {X 0,Y 523.945,Z 214.216,A -85,B 0,C 180,E1 -4635.31,E2 -4635.31} C_VEL
LIN {X 0,Y 523.955,Z 214.223,A -85,B 0,C 180,E1 -4638.69,E2 -4638.69} C_VEL
LIN {X 0,Y 523.917,Z 214.221,A -85,B 0,C 180,E1 -4641.081,E2 -4641.081} C_VEL
LIN {X 0,Y 523.897,Z 214.221,A -85,B 0,C 180,E1 -4643.825,E2 -4643.825} C_VEL
LIN {X 0,Y 523.943,Z 214.224,A -85,B 0,C 180,E1 -4646.635,E2 -4646.635} C_VEL
LIN {X 0,Y 523.957,Z 214.214,A -85,B 0,C 180,E1 -4649.356,E2 -4649.356} C_VEL
LIN {X 0,Y 523.973,Z 214.215,A -85,B 0,C 180,E1 -4652.282,E2 -4652.282} C_VEL
LIN {X 0,Y 523.909,Z 214.219,A -85,B 0,C 180,E1 -4655.427,E2 -4655.427} C_VEL
LIN {X 0,Y 523.939,Z 214.216,A -85,B 0,C 180,E1 -4657.939,E2 -4657.939} C_VEL
LIN {X 0,Y 523.971,Z 214.217,A -85,B 0,C 180,E1 -4660.408,E2 -4660.408} C_VEL
LIN {X 0,Y 523.946,Z 214.221,A -85,B 0,C 180,E1 -4662.836,E2 -4662.836} C_VEL
LIN {X 0,Y 523.969,Z 214.213,A -85,B 0,C 180,E1 -4665.235,E2 -4665.235} C_VEL
LIN {X 0,Y 524.014,Z 214.212,A -85,B 0,C 180,E1 -4668.394,E2 -4668.394} C_VEL
LIN {X 0,Y 523.988,Z 214.209,A -85,B 0,C 180,E1 -4671.516,E2 -4671.516} C_VEL
LIN {X 0,Y 524.078,Z 214.208,A -85,B 0,C 180,E1 -4674.614,E2 -4674.614} C_VEL
LIN {X 0,Y 524.111,Z 214.194,A -85,B 0,C 180,E1 -4677.694,E2 -4677.694} C_VEL
LIN {X 0,Y 524.122,Z 214.199,A -85,B 0,C 180,E1 -4680.768,E2 -4680.768} C_VEL
LIN {X 0,Y 524.042,Z 214.205,A -85,B 0,C 180,E1 -4683.075,E2 -4683.075} C_VEL
LIN {X 0,Y 524.044,Z 214.205,A -85,B 0,C 180,E1 -4686.159,E2 -4686.159} C_VEL
LIN {X 0,Y 524,Z 214.215,A -85,B 0,C 180,E1 -4688.484,E2 -4688.484} C_VEL
LIN {X 0,Y 524.001,Z 214.208,A -85,B 0,C 180,E1 -4691.738,E2 -4691.738} C_VEL
LIN {X 0,Y 523.995,Z 214.211,A -85,B 0,C 180,E1 -4695.053,E2 -4695.053} C_VEL
LIN {X 0,Y 523.948,Z 214.216,A -85,B 0,C 180,E1 -4697.97,E2 -4697.97} C_VEL
LIN {X 0,Y 523.973,Z 214.218,A -85,B 0,C 180,E1 -4700.41,E2 -4700.41} C_VEL
LIN {X 0,Y 523.911,Z 214.223,A -85,B 0,C 180,E1 -4702.894,E2 -4702.894} C_VEL
LIN {X 0,Y 523.935,Z 214.216,A -85,B 0,C 180,E1 -4705.42,E2 -4705.42} C_VEL
LIN {X 0,Y 523.918,Z 214.22,A -85,B 0,C 180,E1 -4708.002,E2 -4708.002} C_VEL
LIN {X 0,Y 523.945,Z 214.22,A -85,B 0,C 180,E1 -4710.855,E2 -4710.855} C_VEL
LIN {X 0,Y 523.93,Z 214.217,A -85,B 0,C 180,E1 -4713.73,E2 -4713.73} C_VEL
LIN {X 0,Y 523.899,Z 214.227,A -85,B 0,C 180,E1 -4716.401,E2 -4716.401} C_VEL
LIN {X 0,Y 523.914,Z 214.221,A -85,B 0,C 180,E1 -4719.085,E2 -4719.085} C_VEL
LIN {X 0,Y 523.941,Z 214.218,A -85,B 0,C 180,E1 -4722.12,E2 -4722.12} C_VEL
LIN {X 0,Y 523.941,Z 214.216,A -85,B 0,C 180,E1 -4725.311,E2 -4725.311} C_VEL
LIN {X 0,Y 523.954,Z 214.221,A -85,B 0,C 180,E1 -4728.69,E2 -4728.69} C_VEL
LIN {X 0,Y 523.916,Z 214.22,A -85,B 0,C 180,E1 -4731.081,E2 -4731.081} C_VEL
LIN {X 0,Y 523.896,Z 214.221,A -85,B 0,C 180,E1 -4733.825,E2 -4733.825} C_VEL
LIN {X 0,Y 523.943,Z 214.223,A -85,B 0,C 180,E1 -4736.636,E2 -4736.636} C_VEL
LIN {X 0,Y 523.95,Z 214.214,A -85,B 0,C 180,E1 -4739.355,E2 -4739.355} C_VEL
LIN {X 0,Y 523.973,Z 214.218,A -85,B 0,C 180,E1 -4742.283,E2 -4742.283} C_VEL
LIN {X 0,Y 523.91,Z 214.221,A -85,B 0,C 180,E1 -4745.427,E2 -4745.427} C_VEL
LIN {X 0,Y 523.935,Z 214.343,A -85,B 0,C 180,E1 -4745.918,E2 -4745.918} C_VEL
LIN {X 0,Y 525.264,Z 221.657,A -85,B 0,C 180,E1 -4747.169,E2 -4747.169} C_VEL
LIN {X 0,Y 524.937,Z 238.229,A -85,B 0,C 180,E1 -4749.834,E2 -4749.834} C_VEL
LIN {X 0,Y 524.555,Z 254.763,A -85,B 0,C 180,E1 -4752.455,E2 -4752.455} C_VEL
LIN {X 0,Y 524.261,Z 269.968,A -85,B 0,C 180,E1 -4754.84,E2 -4754.84} C_VEL
LIN {X 0,Y 525.932,Z 281.164,A -85,B 0,C 180,E1 -4755.047,E2 -4755.047} C_VEL
LIN {X 0,Y 525.508,Z 378.076,A -85,B 0,C 180,E1 -4756.391,E2 -4756.391} C_VEL
LIN {X 0,Y 525.272,Z 391.376,A -85,B 0,C 180,E1 -4756.73,E2 -4756.73} C_VEL
LIN {X 0,Y 525.05,Z 403.556,A -85,B 0,C 180,E1 -4757.191,E2 -4757.191} C_VEL
LIN {X 0,Y 524.743,Z 415.904,A -85,B 0,C 180,E1 -4757.826,E2 -4757.826} C_VEL
LIN {X 0,Y 524.531,Z 427.453,A -85,B 0,C 180,E1 -4758.602,E2 -4758.602} C_VEL
LIN {X 0,Y 524.229,Z 437.902,A -85,B 0,C 180,E1 -4759.475,E2 -4759.475} C_VEL
LIN {X 0,Y 523.979,Z 446.445,A -85,B 0,C 180,E1 -4760.348,E2 -4760.348} C_VEL
LIN {X 0,Y 523.799,Z 454.328,A -85,B 0,C 180,E1 -4761.318,E2 -4761.318} C_VEL
LIN {X 0,Y 523.597,Z 462.026,A -85,B 0,C 180,E1 -4762.48,E2 -4762.48} C_VEL
LIN {X 0,Y 523.478,Z 469.123,A -85,B 0,C 180,E1 -4763.834,E2 -4763.834} C_VEL
LIN {X 0,Y 523.383,Z 473.843,A -85,B 0,C 180,E1 -4764.993,E2 -4764.993} C_VEL
LIN {X 0,Y 523.443,Z 477.452,A -85,B 0,C 180,E1 -4766.151,E2 -4766.151} C_VEL
LIN {X 0,Y 523.367,Z 479.31,A -85,B 0,C 180,E1 -4766.921,E2 -4766.921} C_VEL
LIN {X 0,Y 523.335,Z 480.704,A -85,B 0,C 180,E1 -4767.691,E2 -4767.691} C_VEL
LIN {X 0,Y 523.251,Z 482.305,A -85,B 0,C 180,E1 -4769.23,E2 -4769.23} C_VEL
LIN {X 0,Y 523.249,Z 482.521,A -85,B 0,C 180,E1 -4770,E2 -4770} C_VEL
LIN {X 0,Y 523.274,Z 481.698,A -85,B 0,C 180,E1 -4771.539,E2 -4771.539} C_VEL
LIN {X 0,Y 523.335,Z 480.705,A -85,B 0,C 180,E1 -4772.309,E2 -4772.309} C_VEL
LIN {X 0,Y 523.367,Z 479.311,A -85,B 0,C 180,E1 -4773.079,E2 -4773.079} C_VEL
LIN {X 0,Y 523.423,Z 476.377,A -85,B 0,C 180,E1 -4774.235,E2 -4774.235} C_VEL
LIN {X 0,Y 523.461,Z 472.405,A -85,B 0,C 180,E1 -4775.393,E2 -4775.393} C_VEL
LIN {X 0,Y 523.538,Z 466.328,A -85,B 0,C 180,E1 -4776.739,E2 -4776.739} C_VEL
LIN {X 0,Y 523.662,Z 459.618,A -85,B 0,C 180,E1 -4777.907,E2 -4777.907} C_VEL
LIN {X 0,Y 523.855,Z 451.334,A -85,B 0,C 180,E1 -4779.07,E2 -4779.07} C_VEL
LIN {X 0,Y 524.06,Z 442.843,A -85,B 0,C 180,E1 -4780.04,E2 -4780.04} C_VEL
LIN {X 0,Y 524.36,Z 432.351,A -85,B 0,C 180,E1 -4781.011,E2 -4781.011} C_VEL
LIN {X 0,Y 524.635,Z 422.168,A -85,B 0,C 180,E1 -4781.775,E2 -4781.775} C_VEL
LIN {X 0,Y 524.902,Z 410.593,A -85,B 0,C 180,E1 -4782.468,E2 -4782.468} C_VEL
